METHOD metGetTextListName : STRING
VAR_INPUT
	enTypeOfBacNetFunktionIn		:	enTypeOfBacNetFunktion;
	enTypeOfBacNetTextListIn		:	enTypeOfBacNetTextList;
END_VAR
(* Standart Text *)
IF NOT fbxUseExklTxtList.xValue THEN
	CASE enTypeOfBacNetFunktionIn OF
		(* AT_ANLAGENSCHALTER *)
		enTypeOfBacNetFunktion.Type_Anlagenschalter :
			CASE enTypeOfBacNetTextListIn OF
				enTypeOfBacNetTextList.DESCRIPTION 	:
					metGetTextListName 	:= 'CtaAppBacNetKBOB.TXT_AT_ANLAGENSCHALTER_DESCRIPTION';
				enTypeOfBacNetTextList.ENDING		:
					metGetTextListName 	:= 'CtaAppBacNetKBOB.TXT_AT_ANLAGENSCHALTER_ENDING';
				enTypeOfBacNetTextList.EVENTMESSAGE :
					metGetTextListName 	:= 'CtaAppBacNetKBOB.TXT_AT_ANLAGENSCHALTER_EVENTMESSAGE';
				enTypeOfBacNetTextList.NC			:
					metGetTextListName 	:= 'CtaAppBacNetKBOB.TXT_AT_ANLAGENSCHALTER_NC';
				enTypeOfBacNetTextList.PRESENTVALUE	:
					metGetTextListName	:=	'CtaAppBacNetKBOB.TXT_AT_ANLAGENSCHALTER_PRESV';
				ELSE
					metGetTextListName	:= '';
			END_CASE
		(* AT_ANTRIEB_STETIG *)
		enTypeOfBacNetFunktion.Type_AntriebStetig :
			CASE enTypeOfBacNetTextListIn OF
				enTypeOfBacNetTextList.DESCRIPTION 	:
					metGetTextListName	:= 	'CtaAppBacNetKBOB.TXT_AT_ANTRIEB_STETIG_DESCRIPTION';
				enTypeOfBacNetTextList.ENDING		:
					metGetTextListName	:= 	'CtaAppBacNetKBOB.TXT_AT_ANTRIEB_STETIG_ENDING';
				enTypeOfBacNetTextList.EVENTMESSAGE :
					metGetTextListName	:= 	'CtaAppBacNetKBOB.TXT_AT_ANTRIEB_STETIG_EVENTMESSAGE';
				enTypeOfBacNetTextList.NC			:
					metGetTextListName	:=	'CtaAppBacNetKBOB.TXT_AT_ANTRIEB_STETIG_NC';
				enTypeOfBacNetTextList.PRESENTVALUE	:
					metGetTextListName	:=	'CtaAppBacNetKBOB.TXT_AT_ANTRIEB_STETIG_PRESV';
				ELSE
					metGetTextListName	:= '';
			END_CASE;	
		(* AT_MESSWERTGEBER_BINAR *)
		enTypeOfBacNetFunktion.Type_MesswertgeberBinär :
			CASE enTypeOfBacNetTextListIn OF
				enTypeOfBacNetTextList.DESCRIPTION 	:
					metGetTextListName	:= 	'CtaAppBacNetKBOB.TXT_AT_MESSWERTGEBER_BINAR_DESCRIPTION';
				enTypeOfBacNetTextList.ENDING		:
					metGetTextListName	:= 	'CtaAppBacNetKBOB.TXT_AT_MESSWERTGEBER_BINAR_ENDING';
				enTypeOfBacNetTextList.EVENTMESSAGE :
					metGetTextListName	:= 	'CtaAppBacNetKBOB.TXT_AT_MESSWERTGEBER_BINAR_EVENTMESSAGE';
				enTypeOfBacNetTextList.NC			:
					metGetTextListName	:=	'CtaAppBacNetKBOB.TXT_AT_MESSWERTGEBER_BINAR_NC';
				enTypeOfBacNetTextList.PRESENTVALUE	:
					metGetTextListName	:=	'CtaAppBacNetKBOB.TXT_AT_MESSWERTGEBER_BINAR_PRESV';
				ELSE
					metGetTextListName	:= '';
			END_CASE;
		(* AT_MESSWERTGEBER_STETIG *)
		enTypeOfBacNetFunktion.Type_MesswertgeberStetig :
			CASE enTypeOfBacNetTextListIn OF
				enTypeOfBacNetTextList.DESCRIPTION 	:
					metGetTextListName	:= 	'CtaAppBacNetKBOB.TXT_AT_MESSWERTGEBER_STETIG_DESCRIPTION';
				enTypeOfBacNetTextList.ENDING		:
					metGetTextListName	:= 	'CtaAppBacNetKBOB.TXT_AT_MESSWERTGEBER_STETIG_ENDING';
				enTypeOfBacNetTextList.EVENTMESSAGE :
					metGetTextListName	:= 	'CtaAppBacNetKBOB.TXT_AT_MESSWERTGEBER_STETIG_EVENTMESSAGE';
				enTypeOfBacNetTextList.NC			:
					metGetTextListName	:=	'CtaAppBacNetKBOB.TXT_AT_MESSWERTGEBER_STETIG_NC';
				enTypeOfBacNetTextList.PRESENTVALUE	:
					metGetTextListName	:=	'CtaAppBacNetKBOB.TXT_AT_MESSWERTGEBER_STETIG_PRESV';
				ELSE
					metGetTextListName	:= '';
			END_CASE;
		(* AT_AUTOMATIONSSTATION *)
		enTypeOfBacNetFunktion.Type_Automationsstation :
			CASE enTypeOfBacNetTextListIn OF
				enTypeOfBacNetTextList.DESCRIPTION 	:
					metGetTextListName	:= 	'CtaAppBacNetKBOB.TXT_AT_AUTOMATIONSSTATION_DESCRIPTION';
				enTypeOfBacNetTextList.ENDING		:
					metGetTextListName	:= 	'CtaAppBacNetKBOB.TXT_AT_AUTOMATIONSSTATION_ENDING';
				enTypeOfBacNetTextList.EVENTMESSAGE :
					metGetTextListName	:= 	'CtaAppBacNetKBOB.TXT_AT_AUTOMATIONSSTATION_EVENTMESSAGE';
				enTypeOfBacNetTextList.NC			:
					metGetTextListName	:=	'CtaAppBacNetKBOB.TXT_AT_AUTOMATIONSSTATION_NC';
				enTypeOfBacNetTextList.PRESENTVALUE	:
					metGetTextListName	:=	'CtaAppBacNetKBOB.TXT_AT_AUTOMATIONSSTATION_PRESV';
				ELSE
					metGetTextListName	:= '';
			END_CASE;
		(* AT_ANLAGEFUNKTION *)
		enTypeOfBacNetFunktion.Type_Anlagefunktion :
			CASE enTypeOfBacNetTextListIn OF
				enTypeOfBacNetTextList.DESCRIPTION 	:
					metGetTextListName	:= 	'CtaAppBacNetKBOB.TXT_AT_ANLAGEFUNKTION_DESCRIPTION';
				enTypeOfBacNetTextList.ENDING		:
					metGetTextListName	:= 	'CtaAppBacNetKBOB.TXT_AT_ANLAGEFUNKTION_ENDING';
				enTypeOfBacNetTextList.EVENTMESSAGE :
					metGetTextListName	:= 	'CtaAppBacNetKBOB.TXT_AT_ANLAGEFUNKTION_EVENTMESSAGE';
				enTypeOfBacNetTextList.NC			:
					metGetTextListName	:=	'CtaAppBacNetKBOB.TXT_AT_ANLAGEFUNKTION_NC';
				enTypeOfBacNetTextList.PRESENTVALUE	:
					metGetTextListName	:=	'CtaAppBacNetKBOB.TXT_AT_ANLAGEFUNKTION_PRESV';
				ELSE
					metGetTextListName	:= '';
			END_CASE;		
	ELSE
		metGetTextListName := '';	
	END_CASE;
ELSE
	CASE enTypeOfBacNetFunktionIn OF
		(* AT_ANLAGENSCHALTER *)
		enTypeOfBacNetFunktion.Type_Anlagenschalter :
			CASE enTypeOfBacNetTextListIn OF
				enTypeOfBacNetTextList.DESCRIPTION 	:
					metGetTextListName 	:= 'TXT_AT_ANLAGENSCHALTER_DESCRIPTION';
				enTypeOfBacNetTextList.ENDING		:
					metGetTextListName 	:= 'TXT_AT_ANLAGENSCHALTER_ENDING';
				enTypeOfBacNetTextList.EVENTMESSAGE :
					metGetTextListName 	:= 'TXT_AT_ANLAGENSCHALTER_EVENTMESSAGE';
				enTypeOfBacNetTextList.NC			:
					metGetTextListName 	:= 'TXT_AT_ANLAGENSCHALTER_NC';
				enTypeOfBacNetTextList.PRESENTVALUE	:
					metGetTextListName	:=	'TXT_AT_ANLAGENSCHALTER_PRESV';
				ELSE
					metGetTextListName	:= '';
			END_CASE
		(* AT_ANTRIEB_STETIG *)
		enTypeOfBacNetFunktion.Type_AntriebStetig :
			CASE enTypeOfBacNetTextListIn OF
				enTypeOfBacNetTextList.DESCRIPTION 	:
					metGetTextListName	:= 	'TXT_AT_ANTRIEB_STETIG_DESCRIPTION';
				enTypeOfBacNetTextList.ENDING		:
					metGetTextListName	:= 	'TXT_AT_ANTRIEB_STETIG_ENDING';
				enTypeOfBacNetTextList.EVENTMESSAGE :
					metGetTextListName	:= 	'TXT_AT_ANTRIEB_STETIG_EVENTMESSAGE';
				enTypeOfBacNetTextList.NC			:
					metGetTextListName	:=	'TXT_AT_ANTRIEB_STETIG_NC';
				enTypeOfBacNetTextList.PRESENTVALUE	:
					metGetTextListName	:=	'TXT_AT_ANTRIEB_STETIG_PRESV';
				ELSE
					metGetTextListName	:= '';
			END_CASE;	
		(* AT_MESSWERTGEBER_BINAR *)
		enTypeOfBacNetFunktion.Type_MesswertgeberBinär :
			CASE enTypeOfBacNetTextListIn OF
				enTypeOfBacNetTextList.DESCRIPTION 	:
					metGetTextListName	:= 	'TXT_AT_MESSWERTGEBER_BINAR_DESCRIPTION';
				enTypeOfBacNetTextList.ENDING		:
					metGetTextListName	:= 	'TXT_AT_MESSWERTGEBER_BINAR_ENDING';
				enTypeOfBacNetTextList.EVENTMESSAGE :
					metGetTextListName	:= 	'TXT_AT_MESSWERTGEBER_BINAR_EVENTMESSAGE';
				enTypeOfBacNetTextList.NC			:
					metGetTextListName	:=	'TXT_AT_MESSWERTGEBER_BINAR_NC';
				enTypeOfBacNetTextList.PRESENTVALUE	:
					metGetTextListName	:=	'TXT_AT_MESSWERTGEBER_BINAR_PRESV';
				ELSE
					metGetTextListName	:= '';
			END_CASE;
		(* AT_MESSWERTGEBER_STETIG *)
		enTypeOfBacNetFunktion.Type_MesswertgeberStetig :
			CASE enTypeOfBacNetTextListIn OF
				enTypeOfBacNetTextList.DESCRIPTION 	:
					metGetTextListName	:= 	'TXT_AT_MESSWERTGEBER_STETIG_DESCRIPTION';
				enTypeOfBacNetTextList.ENDING		:
					metGetTextListName	:= 	'TXT_AT_MESSWERTGEBER_STETIG_ENDING';
				enTypeOfBacNetTextList.EVENTMESSAGE :
					metGetTextListName	:= 	'TXT_AT_MESSWERTGEBER_STETIG_EVENTMESSAGE';
				enTypeOfBacNetTextList.NC			:
					metGetTextListName	:=	'TXT_AT_MESSWERTGEBER_STETIG_NC';
				enTypeOfBacNetTextList.PRESENTVALUE	:
					metGetTextListName	:=	'TXT_AT_MESSWERTGEBER_STETIG_PRESV';
				ELSE
					metGetTextListName	:= '';
			END_CASE;
		(* AT_AUTOMATIONSSTATION *)
		enTypeOfBacNetFunktion.Type_Automationsstation :
			CASE enTypeOfBacNetTextListIn OF
				enTypeOfBacNetTextList.DESCRIPTION 	:
					metGetTextListName	:= 	'TXT_AT_AUTOMATIONSSTATION_DESCRIPTION';
				enTypeOfBacNetTextList.ENDING		:
					metGetTextListName	:= 	'TXT_AT_AUTOMATIONSSTATION_ENDING';
				enTypeOfBacNetTextList.EVENTMESSAGE :
					metGetTextListName	:= 	'TXT_AT_MESSWERTGEBER_STETIG_EVENTMESSAGE';
				enTypeOfBacNetTextList.NC			:
					metGetTextListName	:=	'TXT_AT_MESSWERTGEBER_STETIG_NC';
				enTypeOfBacNetTextList.PRESENTVALUE	:
					metGetTextListName	:=	'TXT_AT_MESSWERTGEBER_STETIG_PRESV';
				ELSE
					metGetTextListName	:= '';
			END_CASE;
		(* AT_ANLAGEFUNKTION *)
		enTypeOfBacNetFunktion.Type_Anlagefunktion :
			CASE enTypeOfBacNetTextListIn OF
				enTypeOfBacNetTextList.DESCRIPTION 	:
					metGetTextListName	:= 	'TXT_AT_ANLAGEFUNKTION_DESCRIPTION';
				enTypeOfBacNetTextList.ENDING		:
					metGetTextListName	:= 	'TXT_AT_ANLAGEFUNKTION_ENDING';
				enTypeOfBacNetTextList.EVENTMESSAGE :
					metGetTextListName	:= 	'TXT_AT_ANLAGEFUNKTION_EVENTMESSAGE';
				enTypeOfBacNetTextList.NC			:
					metGetTextListName	:=	'TXT_AT_ANLAGEFUNKTION_NC';
				enTypeOfBacNetTextList.PRESENTVALUE	:
					metGetTextListName	:=	'TXT_AT_ANLAGEFUNKTION_PRESV';
				ELSE
					metGetTextListName	:= '';
			END_CASE;		
	ELSE
		metGetTextListName := '';	
	END_CASE;
END_IF;
END_METHOD

PROPERTY proKBOB_REV : enKBOB_REV
GET
proKBOB_REV := fbenBacNetKbobRev.proValue;
END_GET
END_PROPERTY

PROPERTY P_fbenBacNetKbobRev : CtaSysConfig.ITF_INT
GET
P_fbenBacNetKbobRev := fbenBacNetKbobRev;
END_GET
END_PROPERTY

PROPERTY P_fbxEnableBacNet : CtaSysConfig.ITF_BOOL
GET
P_fbxEnableBacNet := fbxEnableBacNet;
END_GET
END_PROPERTY

PROPERTY P_fbxUseAKS : CtaSysConfig.ITF_BOOL
GET
P_fbxUseAKS := fbxUseAKS;
END_GET
END_PROPERTY

PROPERTY P_fbxUseExklTxtList : CtaSysConfig.ITF_BOOL
GET
P_fbxUseExklTxtList := fbxUseExklTxtList;
END_GET
END_PROPERTY

PROPERTY proTimeToOnline : TIME
GET
IF TON_DELAY_START.Q AND uiCountCreatetObj >= uiCountObj THEN
	proTimeToOnline := T#0S;
ELSE
	proTimeToOnline := (TON_DELAY_START.PT - TON_DELAY_START.ET) + ((uiCountObj * T#6S) - (uiCountCreatetObj * T#6S));
END_IF
END_GET
END_PROPERTY

PROPERTY proDestroyBacNetOverrideXmlNode : BOOL
GET
proDestroyBacNetOverrideXmlNode := xDestroyBacNetOverrideNode;
END_GET
END_PROPERTY

PROPERTY proRebootRequired : BOOL
SET
xRebootRequired := proRebootRequired;
END_SET
GET
proRebootRequired := xRebootRequired;
END_GET
END_PROPERTY

METHOD metAddObj
VAR_INPUT
	ITF_OBJ				:	ITF_OBJ_ID_BASE;
END_VAR
IF __QUERYINTERFACE(ITF_OBJ,ITF_OBJ) THEN
	IF __QUERYINTERFACE(ITF_FIRST_OBJ,ITF_FIRST_OBJ) THEN
		IF ITF_FIRST_OBJ.proINextObj = 0 THEN
			ITF_FIRST_OBJ.proINextObj := ITF_OBJ;
		END_IF;
		IF __QUERYINTERFACE(ITF_NEXT_OBJ,ITF_NEXT_OBJ) THEN
			ITF_NEXT_OBJ.proINextObj := ITF_OBJ;
			ITF_NEXT_OBJ := ITF_OBJ;
		ELSE
			ITF_NEXT_OBJ := ITF_OBJ;
		END_IF;
	ELSIF ITF_FIRST_OBJ = 0 THEN
		ITF_FIRST_OBJ := ITF_OBJ;
	END_IF;	
	uiCountObj := uiCountObj + 1;
END_IF
END_METHOD

ACTION BACNETLIBPARACHECK:
{IF defined (variable: WagoTypesBACnet.Parameter.LEN_BACnetDescription)}
	{IF defined (task: PLC_PRG_Task)}
		{ IF hasconstantvalue(WagoTypesBACnet.Parameter.LEN_BACnetDescription,128,<>)}
			{error 'WagoTypesBACnet.Parameter.LEN_BACnetDescription value <> 128'}
		{END_IF}
	{ELSE}
		{info 'CtaAppBacNetKBOB wurde als Bibliothek Compiliert'}
	{END_IF}
{ELSE}
	{error 'WagoTypesBACnet.Parameter.LEN_BACnetDescription not existing'}
{END_IF}
END_ACTION

PROPERTY P_fbdiDeviceId : CtaSysConfig.ITF_DINT
GET
P_fbdiDeviceId := fbdiDeviceId;
END_GET
END_PROPERTY

PROPERTY P_fbxAnsiCodiert : CtaSysConfig.ITF_BOOL
GET
P_fbxAnsiCodiert := fbxAnsiCodiert;
END_GET
END_PROPERTY

END_FUNCTION_BLOCK

// 30 Program Organization Units/FCs/BacNetIni/fcBacNetIni
FUNCTION fcBacNetIni : BOOL
VAR_INPUT
END_VAR
VAR
	stCommand			:	STRING(255);
	RTS_IEC_RESULT		:	SysTypes.RTS_IEC_RESULT;
END_VAR

(* Replace the persistence-delete from false to true *)
stCommand := 'sed -i $'s/persistence-delete=false/persistence-delete=true/$' /home/user/bacnet/config/bacconfig.ini';
SysProcess_Implementation.SysProcessExecuteCommand(stCommand,ADR(RTS_IEC_RESULT));

END_FUNCTION

// 21 Interface/BACNET_PARAMETER/ITF_BACNET_PARAMETER
INTERFACE ITF_BACNET_PARAMETER EXTENDS __System.IQueryinterface

METHOD metGetTextListName : STRING
VAR_INPUT
	enTypeOfBacNetFunktionIn		:	enTypeOfBacNetFunktion;
	enTypeOfBacNetTextListIn		:	enTypeOfBacNetTextList;
END_VAR
END_METHOD

METHOD metRequestDelete : BOOL
END_METHOD

PROPERTY proCreate : Bool
GET
END_GET
END_PROPERTY

PROPERTY proDelete : Bool
GET
END_GET
END_PROPERTY

PROPERTY proInitDone : BOOL
GET
END_GET
END_PROPERTY

PROPERTY proKBOB_REV : enKBOB_REV
GET
END_GET
END_PROPERTY

PROPERTY proUseAKS : BOOL
GET
END_GET
END_PROPERTY

PROPERTY P_fbxEnableBacNet : CtaSysConfig.ITF_BOOL
GET
END_GET
END_PROPERTY

PROPERTY P_fbxUseAKS : CtaSysConfig.ITF_BOOL
GET
END_GET
END_PROPERTY

PROPERTY P_fbxUseExklTxtList : CtaSysConfig.ITF_BOOL
GET
END_GET
END_PROPERTY

PROPERTY P_fbenBacNetKbobRev : CtaSysConfig.ITF_INT
GET
END_GET
END_PROPERTY

PROPERTY proTimeToOnline : TIME
GET
END_GET
END_PROPERTY

METHOD metAddObj
VAR_INPUT
	ITF_OBJ				:	ITF_OBJ_ID_BASE;
END_VAR
END_METHOD

PROPERTY proRebootRequired : BOOL
SET
END_SET
GET
END_GET
END_PROPERTY

PROPERTY proDestroyBacNetOverrideXmlNode : BOOL
GET
END_GET
END_PROPERTY

PROPERTY P_fbdiDeviceId : CtaSysConfig.ITF_DINT
GET
END_GET
END_PROPERTY

PROPERTY P_fbxAnsiCodiert : CtaSysConfig.ITF_BOOL
GET
END_GET
END_PROPERTY

END_INTERFACE

// 30 Program Organization Units/Pou/BAC_NET
PROGRAM BAC_NET
VAR
END_VAR

(* PARAMETER *)
GVL_BACNET.fbBacNetParameter();
(* AT_DEVICE *)
GVL_BACNET.fbAtAutomationsstation();

END_PROGRAM

// 30 Program Organization Units/FBs/AT_FUNKTIONEN/AT_AUTOMATIONSTATION/FB_AT_AUTOMATIONSSTATION
FUNCTION_BLOCK FB_AT_AUTOMATIONSSTATION EXTENDS FB_OBJ_ID_BASE
VAR
	(* BacNet Objects *)
	A_DV_1				:	WagoSysBACnet.FbDevice_small(-1);						// Device
	B_CL_1				:	WagoSysBACnet.FbCalendar_large(-1);                     // Kalender variable Feiertage
	C_CL_2				:	WagoSysBACnet.FbCalendar_large(-1);                     // Kalender Halbe Tage
	D_CL_3				:	WagoSysBACnet.FbCalendar_large(-1);                     // Kalender feste Feiertage
	E_CL_4				:	WagoSysBACnet.FbCalendar_large(-1);                     // Kalender Ferien
	F_EL_1				:	WagoSysBACnet.FbEventLog_large(-1);						// Eventlog
	G_NC_1				:	WagoSysBACnet.FbNotificationClass_large(-1);			// Notification Class  1 Group Sicherheitsalarm
	G_NC_2				:	WagoSysBACnet.FbNotificationClass_large(-1);			// Notification Class  2 Group Sicherheitsalarm
	G_NC_3				:	WagoSysBACnet.FbNotificationClass_large(-1);			// Notification Class  3 Group Sicherheitsalarm
	G_NC_4				:	WagoSysBACnet.FbNotificationClass_large(-1);			// Notification Class  4 Group Sicherheitsalarm
	H_NC_32				:	WagoSysBACnet.FbNotificationClass_large(-1);			// Notification Class 32 Group Sicherheitsalarm
	H_NC_33				:	WagoSysBACnet.FbNotificationClass_large(-1);			// Notification Class 33 Group Sicherheitsalarm
	H_NC_34				:	WagoSysBACnet.FbNotificationClass_large(-1);			// Notification Class 34 Group Sicherheitsalarm
	H_NC_35				:	WagoSysBACnet.FbNotificationClass_large(-1);			// Notification Class 35 Group Sicherheitsalarm
	I_NC_64				:	WagoSysBACnet.FbNotificationClass_large(-1);			// Notification Class 64 Group Sicherheitsalarm
	I_NC_65				:	WagoSysBACnet.FbNotificationClass_large(-1);			// Notification Class 65 Group Sicherheitsalarm
	I_NC_66				:	WagoSysBACnet.FbNotificationClass_large(-1);			// Notification Class 66 Group Sicherheitsalarm
	I_NC_67				:	WagoSysBACnet.FbNotificationClass_large(-1);			// Notification Class 67 Group Sicherheitsalarm
	J_NC_96				:	WagoSysBACnet.FbNotificationClass_large(-1);			// Notification Class 96 Group Sicherheitsalarm
	J_NC_97				:	WagoSysBACnet.FbNotificationClass_large(-1);			// Notification Class 97 Group Sicherheitsalarm
	J_NC_98				:	WagoSysBACnet.FbNotificationClass_large(-1);			// Notification Class 98 Group Sicherheitsalarm
	J_NC_99				:	WagoSysBACnet.FbNotificationClass_large(-1);			// Notification Class 99 Group Sicherheitsalarm
	K_NC_128			:	WagoSysBACnet.FbNotificationClass_large(-1);			// Notification Class 128 Group Sicherheitsalarm
	K_NC_129			:	WagoSysBACnet.FbNotificationClass_large(-1);			// Notification Class 129 Group Sicherheitsalarm
	K_NC_130			:	WagoSysBACnet.FbNotificationClass_large(-1);			// Notification Class 130 Group Sicherheitsalarm
	K_NC_131			:	WagoSysBACnet.FbNotificationClass_large(-1);			// Notification Class 131 Group Sicherheitsalarm
	L_NC_160			:	WagoSysBACnet.FbNotificationClass_large(-1);			// Notification Class 160 Group Sicherheitsalarm
	L_NC_161			:	WagoSysBACnet.FbNotificationClass_large(-1);			// Notification Class 161 Group Sicherheitsalarm
	L_NC_162			:	WagoSysBACnet.FbNotificationClass_large(-1);			// Notification Class 162 Group Sicherheitsalarm
	L_NC_163			:	WagoSysBACnet.FbNotificationClass_large(-1);			// Notification Class 163 Group Sicherheitsalarm
	M_NC_192			:	WagoSysBACnet.FbNotificationClass_large(-1);			// Notification Class 192 Group Sicherheitsalarm
	M_NC_193			:	WagoSysBACnet.FbNotificationClass_large(-1);			// Notification Class 193 Group Sicherheitsalarm
	N_NC_224			:	WagoSysBACnet.FbNotificationClass_large(-1);			// Notification Class 224 Group Sicherheitsalarm
	N_NC_225			:	WagoSysBACnet.FbNotificationClass_large(-1);			// Notification Class 225 Group Sicherheitsalarm	
	O_BV_1				:	WagoSysBACnet.FbBinaryValue_large(-1);					// CPU State
	P_BV_2				:	WagoSysBACnet.FbBinaryValue_large(-1);					// I/O State
	Q_BV_3				:	WagoSysBACnet.FbBinaryValue_large(-1);					// I/O Hand
	R_BV_4				:	WagoSysBACnet.FbBinaryValue_large(-1);					// Heartbeat
	S_BV_5				:	WagoSysBACnet.FbBinaryValue_large(-1);					// BacStack State
	
END_VAR
VAR CONSTANT
	usiAnzBacNetObj	:	USINT	:= 39;
END_VAR

(* Call Base FB*)
SUPER^();
(* Cyclic Action *)
IF xCreatet THEN
	(* DESCTIPTION FIX *)
	metCYCLIC_DESCRIPTION_FIX();
	(* Get Revision *)
	CASE GVL_BACNET.fbBacNetParameter.proKBOB_REV OF
		(* KBOB 2021 V2 *)
		enKBOB_REV.KBOB_REV2021_V2:
			metCYCLIC_KBOB_2021_V2();
		(* KBOB 2017 V1 *)
		enKBOB_REV.KBOB_REV2017_V1:
			metCYCLIC_KBOB_2017_V1();
		(* Default *)
		ELSE
			metCYCLIC_KBOB_2021_V2();
	END_CASE;	
END_IF;

METHOD metCYCLIC_KBOB_2017_V1
VAR_INPUT
END_VAR
(* CPU Overload *)
IF O_BV_1.xIsCreated THEN
	O_BV_1.xPresentValue := WagoSysBACnet.Common.ControllerInfo.ILedStatus.eLedStatus = WagoTypesBACnet.eBACnetLedStatus.LED_BT_WARNING_OVERLOAD;
END_IF;

(* Check if CtaSysIO exist *)
{IF defined (variable:CtaSysIO.GVL_IO.fbIO_Manager.xError) AND defined (variable:CtaSysIO.GVL_IO.fbIO_Manager.xHand)}
	(* I/O State*) 
	IF P_BV_2.xIsCreated THEN
		P_BV_2.xPresentValue := CtaSysIO.GVL_IO.fbIO_Manager.xError;
	END_IF;

(* I/O Hand *)
	IF Q_BV_3.xIsCreated THEN
		Q_BV_3.xPresentValue := CtaSysIO.GVL_IO.fbIO_Manager.xHand;
	END_IF
{ELSE}
	{warning 'FB_AUTOMATIONSSTATION I/O Infos only with CtaSysIO Library'}
{END_IF}

(* BacStack Error *)
IF S_BV_5.xIsCreated THEN
	S_BV_5.xPresentValue := WagoSysBACnet.Common.ControllerInfo.ILedStatus.eLedStatus = WagoTypesBACnet.eBACnetLedStatus.LED_BT_ERROR_INTERNAL;
END_IF;
END_METHOD

METHOD metCYCLIC_KBOB_2021_V2
VAR_INPUT
END_VAR
(* CPU Overload *)
IF O_BV_1.xIsCreated THEN
	O_BV_1.xPresentValue := WagoSysBACnet.Common.ControllerInfo.ILedStatus.eLedStatus = WagoTypesBACnet.eBACnetLedStatus.LED_BT_WARNING_OVERLOAD;
END_IF;

(* Check if CtaSysIO exist *)
{IF defined (variable:CtaSysIO.GVL_IO.fbIO_Manager.xError) AND defined (variable:CtaSysIO.GVL_IO.fbIO_Manager.xHand)}
	(* I/O State*) 
	IF P_BV_2.xIsCreated THEN
		P_BV_2.xPresentValue := CtaSysIO.GVL_IO.fbIO_Manager.xError;
	END_IF;

(* I/O Hand *)
	IF Q_BV_3.xIsCreated THEN
		Q_BV_3.xPresentValue := CtaSysIO.GVL_IO.fbIO_Manager.xHand;
	END_IF
{ELSE}
	{warning 'FB_AUTOMATIONSSTATION I/O Infos only with CtaSysIO Library'}
{END_IF}

(* BacStack Error *)
IF S_BV_5.xIsCreated THEN
	S_BV_5.xPresentValue := WagoSysBACnet.Common.ControllerInfo.ILedStatus.eLedStatus = WagoTypesBACnet.eBACnetLedStatus.LED_BT_ERROR_INTERNAL;
END_IF;
END_METHOD

METHOD metCYCLIC_DESCRIPTION_FIX
VAR_INPUT
END_VAR
(* A_DV_1 *)
IF A_DV_1.xIsCreated THEN
	IF A_DV_1.sDescription <> A_DV_1._sDescription THEN
		A_DV_1.sDescription := A_DV_1._sDescription;
	END_IF;
END_IF;

(* B_CL_1 *)
IF B_CL_1.xIsCreated THEN
	IF B_CL_1.sDescription <> B_CL_1._sDescription THEN
		B_CL_1.sDescription := B_CL_1._sDescription;
	END_IF;
END_IF;

(* C_CL_2 *)
IF C_CL_2.xIsCreated THEN
	IF C_CL_2.sDescription <> C_CL_2._sDescription THEN
		C_CL_2.sDescription := C_CL_2._sDescription;
	END_IF;
END_IF;

(* D_CL_3 *)
IF D_CL_3.xIsCreated THEN
	IF D_CL_3.sDescription <> D_CL_3._sDescription THEN
		D_CL_3.sDescription := D_CL_3._sDescription;
	END_IF;
END_IF;

(* E_CL_4 *)
IF E_CL_4.xIsCreated THEN
	IF E_CL_4.sDescription <> E_CL_4._sDescription THEN
		E_CL_4.sDescription := E_CL_4._sDescription;
	END_IF;
END_IF;

(* F_EL_1 *)
IF F_EL_1.xIsCreated THEN
	IF F_EL_1.sDescription <> F_EL_1._sDescription THEN
		F_EL_1.sDescription := F_EL_1._sDescription;
	END_IF;
END_IF;

(* G_NC_1 *)
IF G_NC_1.xIsCreated THEN
	IF G_NC_1.sDescription <> G_NC_1._sDescription THEN
		G_NC_1.sDescription := G_NC_1._sDescription;
	END_IF;
END_IF;

(* G_NC_2 *)
IF G_NC_2.xIsCreated THEN
	IF G_NC_2.sDescription <> G_NC_2._sDescription THEN
		G_NC_2.sDescription := G_NC_2._sDescription;
	END_IF;
END_IF;

(* G_NC_3 *)
IF G_NC_3.xIsCreated THEN
	IF G_NC_3.sDescription <> G_NC_3._sDescription THEN
		G_NC_3.sDescription := G_NC_3._sDescription;
	END_IF;
END_IF;

(* G_NC_4 *)
IF G_NC_4.xIsCreated THEN
	IF G_NC_4.sDescription <> G_NC_4._sDescription THEN
		G_NC_4.sDescription := G_NC_4._sDescription;
	END_IF;
END_IF;

(* H_NC_32 *)
IF H_NC_32.xIsCreated THEN
	IF H_NC_32.sDescription <> H_NC_32._sDescription THEN
		H_NC_32.sDescription := H_NC_32._sDescription;
	END_IF;
END_IF;

(* H_NC_33 *)
IF H_NC_33.xIsCreated THEN
	IF H_NC_33.sDescription <> H_NC_33._sDescription THEN
		H_NC_33.sDescription := H_NC_33._sDescription;
	END_IF;
END_IF;

(* H_NC_34 *)
IF H_NC_34.xIsCreated THEN
	IF H_NC_34.sDescription <> H_NC_34._sDescription THEN
		H_NC_34.sDescription := H_NC_34._sDescription;
	END_IF;
END_IF;

(* H_NC_35 *)
IF H_NC_35.xIsCreated THEN
	IF H_NC_35.sDescription <> H_NC_35._sDescription THEN
		H_NC_35.sDescription := H_NC_35._sDescription;
	END_IF;
END_IF;

(* I_NC_64 *)
IF I_NC_64.xIsCreated THEN
	IF I_NC_64.sDescription <> I_NC_64._sDescription THEN
		I_NC_64.sDescription := I_NC_64._sDescription;
	END_IF;
END_IF;

(* I_NC_65 *)
IF I_NC_65.xIsCreated THEN
	IF I_NC_65.sDescription <> I_NC_65._sDescription THEN
		I_NC_65.sDescription := I_NC_65._sDescription;
	END_IF;
END_IF;

(* I_NC_66 *)
IF I_NC_66.xIsCreated THEN
	IF I_NC_66.sDescription <> I_NC_66._sDescription THEN
		I_NC_66.sDescription := I_NC_66._sDescription;
	END_IF;
END_IF;

(* I_NC_67 *)
IF I_NC_67.xIsCreated THEN
	IF I_NC_67.sDescription <> I_NC_67._sDescription THEN
		I_NC_67.sDescription := I_NC_67._sDescription;
	END_IF;
END_IF;

(* J_NC_96 *)
IF J_NC_96.xIsCreated THEN
	IF J_NC_96.sDescription <> J_NC_96._sDescription THEN
		J_NC_96.sDescription := J_NC_96._sDescription;
	END_IF;
END_IF;

(* J_NC_97 *)
IF J_NC_97.xIsCreated THEN
	IF J_NC_97.sDescription <> J_NC_97._sDescription THEN
		J_NC_97.sDescription := J_NC_97._sDescription;
	END_IF;
END_IF;

(* J_NC_98 *)
IF J_NC_98.xIsCreated THEN
	IF J_NC_98.sDescription <> J_NC_98._sDescription THEN
		J_NC_98.sDescription := J_NC_98._sDescription;
	END_IF;
END_IF;

(* J_NC_99 *)
IF J_NC_99.xIsCreated THEN
	IF J_NC_99.sDescription <> J_NC_99._sDescription THEN
		J_NC_99.sDescription := J_NC_99._sDescription;
	END_IF;
END_IF;

(* K_NC_128 *)
IF K_NC_128.xIsCreated THEN
	IF K_NC_128.sDescription <> K_NC_128._sDescription THEN
		K_NC_128.sDescription := K_NC_128._sDescription;
	END_IF;
END_IF;

(* K_NC_129 *)
IF K_NC_129.xIsCreated THEN
	IF K_NC_129.sDescription <> K_NC_129._sDescription THEN
		K_NC_129.sDescription := K_NC_129._sDescription;
	END_IF;
END_IF;

(* K_NC_130 *)
IF K_NC_130.xIsCreated THEN
	IF K_NC_130.sDescription <> K_NC_130._sDescription THEN
		K_NC_130.sDescription := K_NC_130._sDescription;
	END_IF;
END_IF;

(* K_NC_131 *)
IF K_NC_131.xIsCreated THEN
	IF K_NC_131.sDescription <> K_NC_131._sDescription THEN
		K_NC_131.sDescription := K_NC_131._sDescription;
	END_IF;
END_IF;

(* L_NC_160 *)
IF L_NC_160.xIsCreated THEN
	IF L_NC_160.sDescription <> L_NC_160._sDescription THEN
		L_NC_160.sDescription := L_NC_160._sDescription;
	END_IF;
END_IF;

(* L_NC_161 *)
IF L_NC_161.xIsCreated THEN
	IF L_NC_161.sDescription <> L_NC_161._sDescription THEN
		L_NC_161.sDescription := L_NC_161._sDescription;
	END_IF;
END_IF;

(* L_NC_162 *)
IF L_NC_162.xIsCreated THEN
	IF L_NC_162.sDescription <> L_NC_162._sDescription THEN
		L_NC_162.sDescription := L_NC_162._sDescription;
	END_IF;
END_IF;

(* L_NC_163 *)
IF L_NC_163.xIsCreated THEN
	IF L_NC_163.sDescription <> L_NC_163._sDescription THEN
		L_NC_163.sDescription := L_NC_163._sDescription;
	END_IF;
END_IF;

(* M_NC_192 *)
IF M_NC_192.xIsCreated THEN
	IF M_NC_192.sDescription <> M_NC_192._sDescription THEN
		M_NC_192.sDescription := M_NC_192._sDescription;
	END_IF;
END_IF;

(* M_NC_193 *)
IF M_NC_193.xIsCreated THEN
	IF M_NC_193.sDescription <> M_NC_193._sDescription THEN
		M_NC_193.sDescription := M_NC_193._sDescription;
	END_IF;
END_IF;

(* N_NC_224 *)
IF N_NC_224.xIsCreated THEN
	IF N_NC_224.sDescription <> N_NC_224._sDescription THEN
		N_NC_224.sDescription := N_NC_224._sDescription;
	END_IF;
END_IF;

(* N_NC_225 *)
IF N_NC_225.xIsCreated THEN
	IF N_NC_225.sDescription <> N_NC_225._sDescription THEN
		N_NC_225.sDescription := N_NC_225._sDescription;
	END_IF;
END_IF;

(* O_BV_1 *)
IF O_BV_1.xIsCreated THEN
	IF O_BV_1.sDescription <> O_BV_1._sDescription THEN
		O_BV_1.sDescription := O_BV_1._sDescription;
	END_IF;
END_IF;

(* P_BV_2 *)
IF P_BV_2.xIsCreated THEN
	IF P_BV_2.sDescription <> P_BV_2._sDescription THEN
		P_BV_2.sDescription := P_BV_2._sDescription;
	END_IF;
END_IF;

(* Q_BV_3 *)
IF Q_BV_3.xIsCreated THEN
	IF Q_BV_3.sDescription <> Q_BV_3._sDescription THEN
		Q_BV_3.sDescription := Q_BV_3._sDescription;
	END_IF;
END_IF;

(* R_BV_4 *)
IF R_BV_4.xIsCreated THEN
	IF R_BV_4.sDescription <> R_BV_4._sDescription THEN
		R_BV_4.sDescription := R_BV_4._sDescription;
	END_IF;
END_IF;

(* S_BV_5 *)
IF S_BV_5.xIsCreated THEN
	IF S_BV_5.sDescription <> S_BV_5._sDescription THEN
		S_BV_5.sDescription := S_BV_5._sDescription;
	END_IF;
END_IF;
END_METHOD

(*FB_Exit muss explizit implementiert werden. Wenn es eine Implementierung gibt, dann wird 
die Methode aufgerufen, bevor die Steuerung den Code der Funktionsbaustein-Instanz entfernt
(impliziter Aufruf. Der Rückgabewert wird nicht ausgewertet.*)
METHOD FB_Exit : BOOL
VAR_INPUT
	(* TRUE: Die Exit-Methode wird aufgerufen, um die Instanz zu verlassen, die hinterher kopiert wird Online-Change).  *)
	bInCopyCode	: BOOL;
END_VAR
(* A_DV_1 *)
IF A_DV_1.xIsCreated THEN
	A_DV_1.Delete();
END_IF;

(* B_CL_1 *)
IF B_CL_1.xIsCreated THEN
	B_CL_1.Delete();
END_IF;

(* C_CL_2 *)
IF C_CL_2.xIsCreated THEN
	C_CL_2.Delete();
END_IF;

(* D_CL_3 *)
IF D_CL_3.xIsCreated THEN
	D_CL_3.Delete();
END_IF;

(* E_CL_4 *)
IF E_CL_4.xIsCreated THEN
	E_CL_4.Delete();
END_IF;

(* F_EL_1 *)
IF F_EL_1.xIsCreated THEN
	F_EL_1.Delete();
END_IF;

(* G_NC_1 *)
IF G_NC_1.xIsCreated THEN
	G_NC_1.Delete();
END_IF;

(* G_NC_2 *)
IF G_NC_2.xIsCreated THEN
	G_NC_2.Delete();
END_IF;

(* G_NC_3 *)
IF G_NC_3.xIsCreated THEN
	G_NC_3.Delete();
END_IF;

(* G_NC_4 *)
IF G_NC_4.xIsCreated THEN
	G_NC_4.Delete();
END_IF;

(* H_NC_32 *)
IF H_NC_32.xIsCreated THEN
	H_NC_32.Delete();
END_IF;

(* H_NC_33 *)
IF H_NC_33.xIsCreated THEN
	H_NC_33.Delete();
END_IF;

(* H_NC_34 *)
IF H_NC_34.xIsCreated THEN
	H_NC_34.Delete();
END_IF;

(* H_NC_35 *)
IF H_NC_35.xIsCreated THEN
	H_NC_35.Delete();
END_IF;

(* I_NC_64 *)
IF I_NC_64.xIsCreated THEN
	I_NC_64.Delete();
END_IF;

(* I_NC_65 *)
IF I_NC_65.xIsCreated THEN
	I_NC_65.Delete();
END_IF;

(* I_NC_66 *)
IF I_NC_66.xIsCreated THEN
	I_NC_66.Delete();
END_IF;

(* I_NC_67 *)
IF I_NC_67.xIsCreated THEN
	I_NC_67.Delete();
END_IF;

(* J_NC_96 *)
IF J_NC_96.xIsCreated THEN
	J_NC_96.Delete();
END_IF;

(* J_NC_97 *)
IF J_NC_97.xIsCreated THEN
	J_NC_97.Delete();
END_IF;

(* J_NC_98 *)
IF J_NC_98.xIsCreated THEN
	J_NC_98.Delete();
END_IF;

(* J_NC_99 *)
IF J_NC_99.xIsCreated THEN
	J_NC_99.Delete();
END_IF;

(* K_NC_128 *)
IF K_NC_128.xIsCreated THEN
	K_NC_128.Delete();
END_IF;

(* K_NC_129 *)
IF K_NC_129.xIsCreated THEN
	K_NC_129.Delete();
END_IF;

(* K_NC_130 *)
IF K_NC_130.xIsCreated THEN
	K_NC_130.Delete();
END_IF;

(* K_NC_131 *)
IF K_NC_131.xIsCreated THEN
	K_NC_131.Delete();
END_IF;

(* L_NC_160 *)
IF L_NC_160.xIsCreated THEN
	L_NC_160.Delete();
END_IF;

(* L_NC_161 *)
IF L_NC_161.xIsCreated THEN
	L_NC_161.Delete();
END_IF;

(* L_NC_162 *)
IF L_NC_162.xIsCreated THEN
	L_NC_162.Delete();
END_IF;

(* L_NC_163 *)
IF L_NC_163.xIsCreated THEN
	L_NC_163.Delete();
END_IF;

(* M_NC_192 *)
IF M_NC_192.xIsCreated THEN
	M_NC_192.Delete();
END_IF;

(* M_NC_193 *)
IF M_NC_193.xIsCreated THEN
	M_NC_193.Delete();
END_IF;

(* N_NC_224 *)
IF N_NC_224.xIsCreated THEN
	N_NC_224.Delete();
END_IF;

(* N_NC_225 *)
IF N_NC_225.xIsCreated THEN
	N_NC_225.Delete();
END_IF;

(* O_BV_1 *)
IF O_BV_1.xIsCreated THEN
	O_BV_1.Delete();
END_IF;

(* P_BV_2 *)
IF P_BV_2.xIsCreated THEN
	P_BV_2.Delete();
END_IF;

(* Q_BV_3 *)
IF Q_BV_3.xIsCreated THEN
	Q_BV_3.Delete();
END_IF;

(* R_BV_4 *)
IF R_BV_4.xIsCreated THEN
	R_BV_4.Delete();
END_IF;

(* S_BV_5 *)
IF S_BV_5.xIsCreated THEN
	S_BV_5.Delete();
END_IF;
END_METHOD

METHOD metDELETE : BOOL
VAR_INPUT
END_VAR
VAR
	oStatus		:	WagoSysErrorBase.FbResult;
END_VAR
(* A_DV_1 *)
IF A_DV_1.xIsCreated THEN
	A_DV_1.Delete();
END_IF;

(* B_CL_1 *)
IF B_CL_1.xIsCreated THEN
	B_CL_1.Delete();
END_IF;

(* C_CL_2 *)
IF C_CL_2.xIsCreated THEN
	C_CL_2.Delete();
END_IF;

(* D_CL_3 *)
IF D_CL_3.xIsCreated THEN
	D_CL_3.Delete();
END_IF;

(* E_CL_4 *)
IF E_CL_4.xIsCreated THEN
	E_CL_4.Delete();
END_IF;

(* F_EL_1 *)
IF F_EL_1.xIsCreated THEN
	F_EL_1.Delete();
END_IF;

(* G_NC_1 *)
IF G_NC_1.xIsCreated THEN
	G_NC_1.Delete();
END_IF;

(* G_NC_2 *)
IF G_NC_2.xIsCreated THEN
	G_NC_2.Delete();
END_IF;

(* G_NC_3 *)
IF G_NC_3.xIsCreated THEN
	G_NC_3.Delete();
END_IF;

(* G_NC_4 *)
IF G_NC_4.xIsCreated THEN
	G_NC_4.Delete();
END_IF;

(* H_NC_32 *)
IF H_NC_32.xIsCreated THEN
	H_NC_32.Delete();
END_IF;

(* H_NC_33 *)
IF H_NC_33.xIsCreated THEN
	H_NC_33.Delete();
END_IF;

(* H_NC_34 *)
IF H_NC_34.xIsCreated THEN
	H_NC_34.Delete();
END_IF;

(* H_NC_35 *)
IF H_NC_35.xIsCreated THEN
	H_NC_35.Delete();
END_IF;

(* I_NC_64 *)
IF I_NC_64.xIsCreated THEN
	I_NC_64.Delete();
END_IF;

(* I_NC_65 *)
IF I_NC_65.xIsCreated THEN
	I_NC_65.Delete();
END_IF;

(* I_NC_66 *)
IF I_NC_66.xIsCreated THEN
	I_NC_66.Delete();
END_IF;

(* I_NC_67 *)
IF I_NC_67.xIsCreated THEN
	I_NC_67.Delete();
END_IF;

(* J_NC_96 *)
IF J_NC_96.xIsCreated THEN
	J_NC_96.Delete();
END_IF;

(* J_NC_97 *)
IF J_NC_97.xIsCreated THEN
	J_NC_97.Delete();
END_IF;

(* J_NC_98 *)
IF J_NC_98.xIsCreated THEN
	J_NC_98.Delete();
END_IF;

(* J_NC_99 *)
IF J_NC_99.xIsCreated THEN
	J_NC_99.Delete();
END_IF;

(* K_NC_128 *)
IF K_NC_128.xIsCreated THEN
	K_NC_128.Delete();
END_IF;

(* K_NC_129 *)
IF K_NC_129.xIsCreated THEN
	K_NC_129.Delete();
END_IF;

(* K_NC_130 *)
IF K_NC_130.xIsCreated THEN
	K_NC_130.Delete();
END_IF;

(* K_NC_131 *)
IF K_NC_131.xIsCreated THEN
	K_NC_131.Delete();
END_IF;

(* L_NC_160 *)
IF L_NC_160.xIsCreated THEN
	L_NC_160.Delete();
END_IF;

(* L_NC_161 *)
IF L_NC_161.xIsCreated THEN
	L_NC_161.Delete();
END_IF;

(* L_NC_162 *)
IF L_NC_162.xIsCreated THEN
	L_NC_162.Delete();
END_IF;

(* L_NC_163 *)
IF L_NC_163.xIsCreated THEN
	L_NC_163.Delete();
END_IF;

(* M_NC_192 *)
IF M_NC_192.xIsCreated THEN
	M_NC_192.Delete();
END_IF;

(* M_NC_193 *)
IF M_NC_193.xIsCreated THEN
	M_NC_193.Delete();
END_IF;

(* N_NC_224 *)
IF N_NC_224.xIsCreated THEN
	N_NC_224.Delete();
END_IF;

(* N_NC_225 *)
IF N_NC_225.xIsCreated THEN
	N_NC_225.Delete();
END_IF;

(* O_BV_1 *)
IF O_BV_1.xIsCreated THEN
	O_BV_1.Delete();
END_IF;

(* P_BV_2 *)
IF P_BV_2.xIsCreated THEN
	P_BV_2.Delete();
END_IF;

(* Q_BV_3 *)
IF Q_BV_3.xIsCreated THEN
	Q_BV_3.Delete();
END_IF;

(* R_BV_4 *)
IF R_BV_4.xIsCreated THEN
	R_BV_4.Delete();
END_IF;

(* S_BV_5 *)
IF S_BV_5.xIsCreated THEN
	S_BV_5.Delete();
END_IF;
(* Delete Struct View *)
IF GVL_BACNET.fbBacNetParameter.proDestroyBacNetOverrideXmlNode THEN
	fcXMLDeleteOverrideNode(fcBacNetIdToIdWitType(TO_DINT(CONCAT(TO_STRING(OBJ_ID_BASE),'1')),WagoTypesBacNet.eBACnetObjectType.BACnet_structured_view));
	fcXMLDeleteStructuredViewFromDevice(fcBacNetIdToIdWitType(TO_DINT(CONCAT(TO_STRING(OBJ_ID_BASE),'1')),WagoTypesBacNet.eBACnetObjectType.BACnet_structured_view));
END_IF;
metDELETE := 	A_DV_1.xIsCreated OR 
				B_CL_1.xIsCreated OR
				C_CL_2.xIsCreated OR				
				E_CL_4.xIsCreated OR
				F_EL_1.xIsCreated OR
				G_NC_1.xIsCreated OR
				G_NC_2.xIsCreated OR
				G_NC_3.xIsCreated OR
				G_NC_4.xIsCreated OR
				H_NC_32.xIsCreated OR
				H_NC_33.xIsCreated OR
				H_NC_34.xIsCreated OR
				H_NC_35.xIsCreated OR
				I_NC_64.xIsCreated OR
				I_NC_65.xIsCreated OR
				I_NC_66.xIsCreated OR
				I_NC_67.xIsCreated OR
				J_NC_96.xIsCreated OR
				J_NC_97.xIsCreated OR
				J_NC_98.xIsCreated OR
				J_NC_99.xIsCreated OR
				K_NC_128.xIsCreated OR
				K_NC_129.xIsCreated OR
				K_NC_130.xIsCreated OR
				K_NC_131.xIsCreated OR
				L_NC_160.xIsCreated OR
				L_NC_161.xIsCreated OR
				L_NC_162.xIsCreated OR
				L_NC_163.xIsCreated OR
				M_NC_192.xIsCreated OR
				M_NC_193.xIsCreated OR
				N_NC_224.xIsCreated OR
				N_NC_225.xIsCreated OR
				O_BV_1.xIsCreated OR
				P_BV_2.xIsCreated OR
				Q_BV_3.xIsCreated OR
				R_BV_4.xIsCreated OR
				S_BV_5.xIsCreated ;
(* Reset Create Case *)
usiCreateCase := 1;
END_METHOD

METHOD metCREATE_KBOB_2017_V1 : BOOL;
VAR_INPUT
END_VAR
VAR
	oStatus		:	WagoSysErrorBase.FbResult;
	usiErrors	:	USINT;
END_VAR
(* Resett *)
usiErrors := 0;	

(* Create Objeccts *)
CASE usiCreateCase OF
	1:	
		usiErrors := usiErrors + TO_USINT(NOT metCreate_A_DV_1());
	2:
		usiErrors := usiErrors + TO_USINT(NOT metCreate_B_CL_1());
	3:	
		usiErrors := usiErrors + TO_USINT(NOT metCreate_C_CL_2());
	4:	
		usiErrors := usiErrors + TO_USINT(NOT metCreate_D_CL_3());
	5:
		usiErrors := usiErrors + TO_USINT(NOT metCreate_E_CL_4());
	6:	
		usiErrors := usiErrors + TO_USINT(NOT metCreate_F_EL_1());
	7:
		usiErrors := usiErrors + TO_USINT(NOT metCreate_G_NC_1());
	8:	
		usiErrors := usiErrors + TO_USINT(NOT metCreate_G_NC_2());
	9:
		usiErrors := usiErrors + TO_USINT(NOT metCreate_G_NC_3());
	10:
		usiErrors := usiErrors + TO_USINT(NOT metCreate_G_NC_4());
	11:	
		usiErrors := usiErrors + TO_USINT(NOT metCreate_H_NC_32());
	12:
		usiErrors := usiErrors + TO_USINT(NOT metCreate_H_NC_33());
	13:
		usiErrors := usiErrors + TO_USINT(NOT metCreate_H_NC_34());
	14:
		usiErrors := usiErrors + TO_USINT(NOT metCreate_H_NC_35());
	15:
		usiErrors := usiErrors + TO_USINT(NOT metCreate_I_NC_64());
	16:
		usiErrors := usiErrors + TO_USINT(NOT metCreate_I_NC_65());
	17:
		usiErrors := usiErrors + TO_USINT(NOT metCreate_I_NC_66());
	18:
		usiErrors := usiErrors + TO_USINT(NOT metCreate_I_NC_67());
	19:
		usiErrors := usiErrors + TO_USINT(NOT metCreate_J_NC_96());
	20:
		usiErrors := usiErrors + TO_USINT(NOT metCreate_J_NC_97());
	21:
		usiErrors := usiErrors + TO_USINT(NOT metCreate_J_NC_98());
	22:
		usiErrors := usiErrors + TO_USINT(NOT metCreate_J_NC_99());
	23:
		usiErrors := usiErrors + TO_USINT(NOT metCreate_K_NC_128());
	24:
		usiErrors := usiErrors + TO_USINT(NOT metCreate_K_NC_129());
	25:
		usiErrors := usiErrors + TO_USINT(NOT metCreate_K_NC_130());
	26:
		usiErrors := usiErrors + TO_USINT(NOT metCreate_K_NC_131());
	27:
		usiErrors := usiErrors + TO_USINT(NOT metCreate_L_NC_160());
	28:
		usiErrors := usiErrors + TO_USINT(NOT metCreate_L_NC_161());
	29:
		usiErrors := usiErrors + TO_USINT(NOT metCreate_L_NC_162());
	30:
		usiErrors := usiErrors + TO_USINT(NOT metCreate_L_NC_163());
	31:
		usiErrors := usiErrors + TO_USINT(NOT metCreate_M_NC_192());
	32:
		usiErrors := usiErrors + TO_USINT(NOT metCreate_M_NC_193());
	33:
		usiErrors := usiErrors + TO_USINT(NOT metCreate_N_NC_224());
	34:
		usiErrors := usiErrors + TO_USINT(NOT metCreate_N_NC_225());
	35:
		usiErrors := usiErrors + TO_USINT(NOT metCreate_O_BV_1());
	36:
		usiErrors := usiErrors + TO_USINT(NOT metCreate_P_BV_2());
	37:
		usiErrors := usiErrors + TO_USINT(NOT metCreate_Q_BV_3());
	38:
		usiErrors := usiErrors + TO_USINT(NOT metCreate_R_BV_4());
	39:
		usiErrors := usiErrors + TO_USINT(NOT metCreate_S_BV_5());
	0: 
		usiCreateCase := 1;
ELSE
	usiCreateCase := 0;
END_CASE;

(* STRUCT VIEW *)
metCREATE_STRUCTVIEW_KBOB_2017_V1();

(* OK = 0*)
metCREATE_KBOB_2017_V1 := NOT TO_BOOL(usiErrors);
END_METHOD

METHOD metCREATE_STRUCTVIEW_KBOB_2017_V1 : BOOL
VAR_INPUT
END_VAR
CASE usiCreateCase OF
	1:
		fcXMLStructuredView(THIS^,A_DV_1.IObjectIdentifier);			
	2:                                                                 
		fcXMLStructuredView(THIS^,B_CL_1.IObjectIdentifier);            
	3:                                                                 
		fcXMLStructuredView(THIS^,C_CL_2.IObjectIdentifier);            
	4:                                                                 
		fcXMLStructuredView(THIS^,D_CL_3.IObjectIdentifier);            
	5:                                                                 
		fcXMLStructuredView(THIS^,E_CL_4.IObjectIdentifier);            
	6:                                                                 
		fcXMLStructuredView(THIS^,F_EL_1.IObjectIdentifier);            
	7:                                                                 
		fcXMLStructuredView(THIS^,G_NC_1.IObjectIdentifier);            
	8:                                                                 
		fcXMLStructuredView(THIS^,G_NC_2.IObjectIdentifier);            
	9:                                                                 
		fcXMLStructuredView(THIS^,G_NC_3.IObjectIdentifier);            
	10:                                                                
		fcXMLStructuredView(THIS^,G_NC_4.IObjectIdentifier);            
	11:                                                                
		fcXMLStructuredView(THIS^,H_NC_32.IObjectIdentifier);           
	12:                                                                
		fcXMLStructuredView(THIS^,H_NC_33.IObjectIdentifier);  
	13:                                                                
		fcXMLStructuredView(THIS^,H_NC_34.IObjectIdentifier);  
	14:                                                                
		fcXMLStructuredView(THIS^,H_NC_35.IObjectIdentifier);           
	15:                                                                
		 fcXMLStructuredView(THIS^,I_NC_64.IObjectIdentifier);           
	16:                                                                
		 fcXMLStructuredView(THIS^,I_NC_65.IObjectIdentifier);           
	17:                                                                
		 fcXMLStructuredView(THIS^,I_NC_66.IObjectIdentifier);           
	18:	                                                               
		 fcXMLStructuredView(THIS^,I_NC_67.IObjectIdentifier);           
	19:                                                                
		 fcXMLStructuredView(THIS^,J_NC_96.IObjectIdentifier);           
	20:                                                                
		 fcXMLStructuredView(THIS^,J_NC_97.IObjectIdentifier);           
	21:                                                                
		 fcXMLStructuredView(THIS^,J_NC_98.IObjectIdentifier);           
	22:                                                                
		 fcXMLStructuredView(THIS^,J_NC_99.IObjectIdentifier);           
	23:                                                                
		 fcXMLStructuredView(THIS^,K_NC_128.IObjectIdentifier);          
	24:                                                                
		 fcXMLStructuredView(THIS^,K_NC_129.IObjectIdentifier);          
	25:                                                                
		 fcXMLStructuredView(THIS^,K_NC_130.IObjectIdentifier);          
	26:                                                                
		 fcXMLStructuredView(THIS^,K_NC_131.IObjectIdentifier);          
	27:                                                                
		 fcXMLStructuredView(THIS^,L_NC_160.IObjectIdentifier);          
	28:                                                                
		 fcXMLStructuredView(THIS^,L_NC_161.IObjectIdentifier);          
	29:                                                                
		 fcXMLStructuredView(THIS^,L_NC_162.IObjectIdentifier);          
	30:                                                                
		 fcXMLStructuredView(THIS^,L_NC_163.IObjectIdentifier);		    
	31:                                                                
		 fcXMLStructuredView(THIS^,M_NC_192.IObjectIdentifier);          
	32:                                                                
		 fcXMLStructuredView(THIS^,M_NC_193.IObjectIdentifier);          
	33:                                                                
		 fcXMLStructuredView(THIS^,N_NC_224.IObjectIdentifier);          
	34:                                                                
		 fcXMLStructuredView(THIS^,N_NC_225.IObjectIdentifier);	        
	35:                                                                
		 fcXMLStructuredView(THIS^,O_BV_1.IObjectIdentifier);            
	36:                                                                
		 fcXMLStructuredView(THIS^,P_BV_2.IObjectIdentifier);            
	37:                                                                
		fcXMLStructuredView(THIS^,Q_BV_3.IObjectIdentifier);            
	38:                                                                
		fcXMLStructuredView(THIS^,R_BV_4.IObjectIdentifier);            
	39:                                                                
		fcXMLStructuredView(THIS^,S_BV_5.IObjectIdentifier);            	                                                               
		fcXMLAddStructuredViewToDevice(THIS^);	                            
	0:                                                                 
		usiCreateCase := 1;                                             
ELSE
	usiCreateCase := 0;
END_CASE
END_METHOD

METHOD metCREATE_KBOB_2021_V2 : BOOL;
VAR_INPUT
END_VAR
VAR
	oStatus		:	WagoSysErrorBase.FbResult;
	usiErrors	:	USINT;
END_VAR
(* Resett *)
usiErrors := 0;	

(* Create Objeccts *)
CASE usiCreateCase OF
	1:	
		usiErrors := usiErrors + TO_USINT(NOT metCreate_A_DV_1());
	2:
		usiErrors := usiErrors + TO_USINT(NOT metCreate_B_CL_1());
	3:	
		usiErrors := usiErrors + TO_USINT(NOT metCreate_C_CL_2());
	4:	
		usiErrors := usiErrors + TO_USINT(NOT metCreate_D_CL_3());
	5:
		usiErrors := usiErrors + TO_USINT(NOT metCreate_E_CL_4());
	6:	
		usiErrors := usiErrors + TO_USINT(NOT metCreate_F_EL_1());
	7:
		usiErrors := usiErrors + TO_USINT(NOT metCreate_G_NC_1());
	8:	
		usiErrors := usiErrors + TO_USINT(NOT metCreate_G_NC_2());
	9:
		usiErrors := usiErrors + TO_USINT(NOT metCreate_G_NC_3());
	10:
		usiErrors := usiErrors + TO_USINT(NOT metCreate_G_NC_4());
	11:	
		usiErrors := usiErrors + TO_USINT(NOT metCreate_H_NC_32());
	12:
		usiErrors := usiErrors + TO_USINT(NOT metCreate_H_NC_33());
	13:
		usiErrors := usiErrors + TO_USINT(NOT metCreate_H_NC_34());
	14:
		usiErrors := usiErrors + TO_USINT(NOT metCreate_H_NC_35());
	15:
		usiErrors := usiErrors + TO_USINT(NOT metCreate_I_NC_64());
	16:
		usiErrors := usiErrors + TO_USINT(NOT metCreate_I_NC_65());
	17:
		usiErrors := usiErrors + TO_USINT(NOT metCreate_I_NC_66());
	18:
		usiErrors := usiErrors + TO_USINT(NOT metCreate_I_NC_67());
	19:
		usiErrors := usiErrors + TO_USINT(NOT metCreate_J_NC_96());
	20:
		usiErrors := usiErrors + TO_USINT(NOT metCreate_J_NC_97());
	21:
		usiErrors := usiErrors + TO_USINT(NOT metCreate_J_NC_98());
	22:
		usiErrors := usiErrors + TO_USINT(NOT metCreate_J_NC_99());
	23:
		usiErrors := usiErrors + TO_USINT(NOT metCreate_K_NC_128());
	24:
		usiErrors := usiErrors + TO_USINT(NOT metCreate_K_NC_129());
	25:
		usiErrors := usiErrors + TO_USINT(NOT metCreate_K_NC_130());
	26:
		usiErrors := usiErrors + TO_USINT(NOT metCreate_K_NC_131());
	27:
		usiErrors := usiErrors + TO_USINT(NOT metCreate_L_NC_160());
	28:
		usiErrors := usiErrors + TO_USINT(NOT metCreate_L_NC_161());
	29:
		usiErrors := usiErrors + TO_USINT(NOT metCreate_L_NC_162());
	30:
		usiErrors := usiErrors + TO_USINT(NOT metCreate_L_NC_163());
	31:
		usiErrors := usiErrors + TO_USINT(NOT metCreate_M_NC_192());
	32:
		usiErrors := usiErrors + TO_USINT(NOT metCreate_M_NC_193());
	33:
		usiErrors := usiErrors + TO_USINT(NOT metCreate_N_NC_224());
	34:
		usiErrors := usiErrors + TO_USINT(NOT metCreate_N_NC_225());
	35:
		usiErrors := usiErrors + TO_USINT(NOT metCreate_O_BV_1());
	36:
		usiErrors := usiErrors + TO_USINT(NOT metCreate_P_BV_2());
	37:
		usiErrors := usiErrors + TO_USINT(NOT metCreate_Q_BV_3());
	38:
		usiErrors := usiErrors + TO_USINT(NOT metCreate_R_BV_4());
	39:
		usiErrors := usiErrors + TO_USINT(NOT metCreate_S_BV_5());
	0: 
		usiCreateCase := 1;
ELSE
	usiCreateCase := 0;
END_CASE;

(* STRUCT VIEW *)
metCREATE_STRUCTVIEW_KBOB_2021_V2();

(* OK = 0*)
metCREATE_KBOB_2021_V2 := NOT TO_BOOL(usiErrors);
END_METHOD

METHOD metCREATE_STRUCTVIEW_KBOB_2021_V2 : BOOL
VAR_INPUT
END_VAR
CASE usiCreateCase OF
	1:
		fcXMLStructuredView(THIS^,A_DV_1.IObjectIdentifier);			
	2:                                                                 
		fcXMLStructuredView(THIS^,B_CL_1.IObjectIdentifier);            
	3:                                                                 
		fcXMLStructuredView(THIS^,C_CL_2.IObjectIdentifier);            
	4:                                                                 
		fcXMLStructuredView(THIS^,D_CL_3.IObjectIdentifier);            
	5:                                                                 
		fcXMLStructuredView(THIS^,E_CL_4.IObjectIdentifier);            
	6:                                                                 
		fcXMLStructuredView(THIS^,F_EL_1.IObjectIdentifier);            
	7:                                                                 
		fcXMLStructuredView(THIS^,G_NC_1.IObjectIdentifier);            
	8:                                                                 
		fcXMLStructuredView(THIS^,G_NC_2.IObjectIdentifier);            
	9:                                                                 
		fcXMLStructuredView(THIS^,G_NC_3.IObjectIdentifier);            
	10:                                                                
		fcXMLStructuredView(THIS^,G_NC_4.IObjectIdentifier);            
	11:                                                                
		fcXMLStructuredView(THIS^,H_NC_32.IObjectIdentifier);           
	12:                                                                
		fcXMLStructuredView(THIS^,H_NC_33.IObjectIdentifier);  
	13:                                                                
		fcXMLStructuredView(THIS^,H_NC_34.IObjectIdentifier);  
	14:                                                                
		fcXMLStructuredView(THIS^,H_NC_35.IObjectIdentifier);           
	15:                                                                
		 fcXMLStructuredView(THIS^,I_NC_64.IObjectIdentifier);           
	16:                                                                
		 fcXMLStructuredView(THIS^,I_NC_65.IObjectIdentifier);           
	17:                                                                
		 fcXMLStructuredView(THIS^,I_NC_66.IObjectIdentifier);           
	18:	                                                               
		 fcXMLStructuredView(THIS^,I_NC_67.IObjectIdentifier);           
	19:                                                                
		 fcXMLStructuredView(THIS^,J_NC_96.IObjectIdentifier);           
	20:                                                                
		 fcXMLStructuredView(THIS^,J_NC_97.IObjectIdentifier);           
	21:                                                                
		 fcXMLStructuredView(THIS^,J_NC_98.IObjectIdentifier);           
	22:                                                                
		 fcXMLStructuredView(THIS^,J_NC_99.IObjectIdentifier);           
	23:                                                                
		 fcXMLStructuredView(THIS^,K_NC_128.IObjectIdentifier);          
	24:                                                                
		 fcXMLStructuredView(THIS^,K_NC_129.IObjectIdentifier);          
	25:                                                                
		 fcXMLStructuredView(THIS^,K_NC_130.IObjectIdentifier);          
	26:                                                                
		 fcXMLStructuredView(THIS^,K_NC_131.IObjectIdentifier);          
	27:                                                                
		 fcXMLStructuredView(THIS^,L_NC_160.IObjectIdentifier);          
	28:                                                                
		 fcXMLStructuredView(THIS^,L_NC_161.IObjectIdentifier);          
	29:                                                                
		 fcXMLStructuredView(THIS^,L_NC_162.IObjectIdentifier);          
	30:                                                                
		 fcXMLStructuredView(THIS^,L_NC_163.IObjectIdentifier);		    
	31:                                                                
		 fcXMLStructuredView(THIS^,M_NC_192.IObjectIdentifier);          
	32:                                                                
		 fcXMLStructuredView(THIS^,M_NC_193.IObjectIdentifier);          
	33:                                                                
		 fcXMLStructuredView(THIS^,N_NC_224.IObjectIdentifier);          
	34:                                                                
		 fcXMLStructuredView(THIS^,N_NC_225.IObjectIdentifier);	        
	35:                                                                
		 fcXMLStructuredView(THIS^,O_BV_1.IObjectIdentifier);            
	36:                                                                
		 fcXMLStructuredView(THIS^,P_BV_2.IObjectIdentifier);            
	37:                                                                
		fcXMLStructuredView(THIS^,Q_BV_3.IObjectIdentifier);            
	38:                                                                
		fcXMLStructuredView(THIS^,R_BV_4.IObjectIdentifier);            
	39:                                                                
		fcXMLStructuredView(THIS^,S_BV_5.IObjectIdentifier);            	                                                               
		fcXMLAddStructuredViewToDevice(THIS^);	                            
	0:                                                                 
		usiCreateCase := 1;                                             
ELSE
	usiCreateCase := 0;
END_CASE
END_METHOD

METHOD metCREATE : BOOL;
VAR_INPUT
END_VAR
VAR
	oStatus		:	WagoSysErrorBase.FbResult;
	usiErrors	:	USINT;
END_VAR
(* Get Revision *)
CASE GVL_BACNET.fbBacNetParameter.proKBOB_REV OF
	(* KBOB 2021 V2 *)
	enKBOB_REV.KBOB_REV2021_V2:
		usiErrors := usiErrors + TO_USINT(NOT metCREATE_KBOB_2021_V2());
	(* KBOB 2017 V1 *)
	enKBOB_REV.KBOB_REV2017_V1:
		usiErrors := usiErrors + TO_USINT(NOT metCREATE_KBOB_2017_V1());
	(* Default *)
	ELSE
		usiErrors := usiErrors + TO_USINT(NOT metCREATE_KBOB_2021_V2());
END_CASE;

(* OK = 0*)
xErrorCreate := TO_BOOL(usiErrors);
metCREATE := NOT TO_BOOL(usiErrors) AND usiCreateCase = usiAnzBacNetObj;
END_METHOD

METHOD metCreate_L_NC_160 : BOOL

VAR

END_VAR
(* L_NC_160*)
IF NOT L_NC_160.xIsCreated THEN
	(* Ziel						UTF8->ASCII						OBJ_NAME_BASE			BacNet Text		Textlistname									BacNet Funktion																	BacNet Textlist type												TextId		*)
	L_NC_160._sObjectName		:=	fcUtfToAscii(Standard.CONCAT(	OBJ_NAME_BASE		,	fcGetBcText(	GVL_BACNET.fbBacNetParameter.metGetTextListName(enTypeOfBacNetFunktionIn := enTypeOfBacNetFunktion.Type_Automationsstation,		enTypeOfBacNetTextListIn := enTypeOfBacNetTextList.ENDING		),	'L_NC_160')));
	L_NC_160._sDescription	:= 	fcUtfToAscii(Standard.CONCAT(	OBJ_NAME_DESCRIPTION,	fcGetBcText(	GVL_BACNET.fbBacNetParameter.metGetTextListName(enTypeOfBacNetFunktionIn := enTypeOfBacNetFunktion.Type_Automationsstation,		enTypeOfBacNetTextListIn := enTypeOfBacNetTextList.DESCRIPTION	),	'L_NC_160')));
	(* Create Id from Base Id and Object Nr (Last nummber of Name *)	
	L_NC_160.Create(diInstance := 160);
	(* Check if Created *)
	IF L_NC_160.xIsCreated THEN
		(* Set Group *)
		L_NC_160.setPropertyGroup(WagoTypesBacNet.eBACnetPropertyIdentifier.PROP_DESCRIPTION							,WagoTypesBacNet.eBACnetPropertyUpdateGroup.GROUP_CYCLIC);
		
		(* Set Ack Req *)
		L_NC_160.IAckRequired.xToOffNormal	:= FALSE;
		L_NC_160.IAckRequired.xToFault		:= FALSE;
		L_NC_160.IAckRequired.xToNormal		:= FALSE;
		
		(* Ziel												UTF8->ASCII		BacNet Text		Textlistname									BacNet Funktion																	BacNet Textlist type												TextId		*)
		L_NC_160.IEventMessageTextsConfig.sToOffNormal	:=	fcUtfToAscii(	fcGetBcText(	GVL_BACNET.fbBacNetParameter.metGetTextListName(enTypeOfBacNetFunktionIn := enTypeOfBacNetFunktion.Type_Automationsstation,		enTypeOfBacNetTextListIn := enTypeOfBacNetTextList.EVENTMESSAGE	),	'L_NC_160_ToOffNormal'	));		
		L_NC_160.IEventMessageTextsConfig.sToFault		:=	fcUtfToAscii(	fcGetBcText(	GVL_BACNET.fbBacNetParameter.metGetTextListName(enTypeOfBacNetFunktionIn := enTypeOfBacNetFunktion.Type_Automationsstation,		enTypeOfBacNetTextListIn := enTypeOfBacNetTextList.EVENTMESSAGE	),	'L_NC_160_ToFault'		));		
		L_NC_160.IEventMessageTextsConfig.sToNormal		:=	fcUtfToAscii(	fcGetBcText(	GVL_BACNET.fbBacNetParameter.metGetTextListName(enTypeOfBacNetFunktionIn := enTypeOfBacNetFunktion.Type_Automationsstation,		enTypeOfBacNetTextListIn := enTypeOfBacNetTextList.EVENTMESSAGE	),	'L_NC_160_ToNormal'		));		
		
		(* Notification Class & Type *)
		L_NC_160.udiNotificationClass					:=  160;	
		L_NC_160.eNotifyType							:= 	WagoTypesBACnet.eBACnetNotifyType.NOTIFY_TYPE_ALARM;
		(* Ziel												Convert			BacNet Text		Textlistname									BacNet Funktion																	BacNet Textlist type												TextId		*)	
		L_NC_160.IPriority.usiToOffNormal				:= 	TO_USINT(fcUtfToAscii(	fcGetBcText(	GVL_BACNET.fbBacNetParameter.metGetTextListName(enTypeOfBacNetFunktionIn := enTypeOfBacNetFunktion.Type_Automationsstation,		enTypeOfBacNetTextListIn := enTypeOfBacNetTextList.NC	),	'L_NC_160_Prio_ToOffNormal'	)));	
		L_NC_160.IPriority.usiToFault					:= 	TO_USINT(fcUtfToAscii(	fcGetBcText(	GVL_BACNET.fbBacNetParameter.metGetTextListName(enTypeOfBacNetFunktionIn := enTypeOfBacNetFunktion.Type_Automationsstation,		enTypeOfBacNetTextListIn := enTypeOfBacNetTextList.NC	),	'L_NC_160_Prio_ToFault'		)));	
		L_NC_160.IPriority.usiToNormal					:= 	TO_USINT(fcUtfToAscii(	fcGetBcText(	GVL_BACNET.fbBacNetParameter.metGetTextListName(enTypeOfBacNetFunktionIn := enTypeOfBacNetFunktion.Type_Automationsstation,		enTypeOfBacNetTextListIn := enTypeOfBacNetTextList.NC	),	'L_NC_160_Prio_ToNormal'		)));	
		
	ELSE
		L_NC_160.Delete();
	END_IF;
	(* Get Status *)
	metCreate_L_NC_160 := L_NC_160.xIsCreated;	
END_IF;
END_METHOD

METHOD metCreate_L_NC_161 : BOOL

VAR

END_VAR
(* L_NC_161*)
IF NOT L_NC_161.xIsCreated THEN
	(* Ziel						UTF8->ASCII						OBJ_NAME_BASE			BacNet Text		Textlistname									BacNet Funktion																	BacNet Textlist type												TextId		*)
	L_NC_161._sObjectName		:=	fcUtfToAscii(Standard.CONCAT(	OBJ_NAME_BASE		,	fcGetBcText(	GVL_BACNET.fbBacNetParameter.metGetTextListName(enTypeOfBacNetFunktionIn := enTypeOfBacNetFunktion.Type_Automationsstation,		enTypeOfBacNetTextListIn := enTypeOfBacNetTextList.ENDING		),	'L_NC_161')));
	L_NC_161._sDescription	:= 	fcUtfToAscii(Standard.CONCAT(	OBJ_NAME_DESCRIPTION,	fcGetBcText(	GVL_BACNET.fbBacNetParameter.metGetTextListName(enTypeOfBacNetFunktionIn := enTypeOfBacNetFunktion.Type_Automationsstation,		enTypeOfBacNetTextListIn := enTypeOfBacNetTextList.DESCRIPTION	),	'L_NC_161')));
	(* Create Id from Base Id and Object Nr (Last nummber of Name *)	
	L_NC_161.Create(diInstance := 161);
	(* Check if Created *)
	IF L_NC_161.xIsCreated THEN
		(* Set Group *)
		L_NC_161.setPropertyGroup(WagoTypesBacNet.eBACnetPropertyIdentifier.PROP_DESCRIPTION							,WagoTypesBacNet.eBACnetPropertyUpdateGroup.GROUP_CYCLIC);
		
		(* Set Ack Req *)
		L_NC_161.IAckRequired.xToOffNormal	:= FALSE;
		L_NC_161.IAckRequired.xToFault		:= TRUE;
		L_NC_161.IAckRequired.xToNormal		:= FALSE;
		
		(* Ziel												UTF8->ASCII		BacNet Text		Textlistname									BacNet Funktion																	BacNet Textlist type												TextId		*)
		L_NC_161.IEventMessageTextsConfig.sToOffNormal	:=	fcUtfToAscii(	fcGetBcText(	GVL_BACNET.fbBacNetParameter.metGetTextListName(enTypeOfBacNetFunktionIn := enTypeOfBacNetFunktion.Type_Automationsstation,		enTypeOfBacNetTextListIn := enTypeOfBacNetTextList.EVENTMESSAGE	),	'L_NC_161_ToOffNormal'	));		
		L_NC_161.IEventMessageTextsConfig.sToFault		:=	fcUtfToAscii(	fcGetBcText(	GVL_BACNET.fbBacNetParameter.metGetTextListName(enTypeOfBacNetFunktionIn := enTypeOfBacNetFunktion.Type_Automationsstation,		enTypeOfBacNetTextListIn := enTypeOfBacNetTextList.EVENTMESSAGE	),	'L_NC_161_ToFault'		));		
		L_NC_161.IEventMessageTextsConfig.sToNormal		:=	fcUtfToAscii(	fcGetBcText(	GVL_BACNET.fbBacNetParameter.metGetTextListName(enTypeOfBacNetFunktionIn := enTypeOfBacNetFunktion.Type_Automationsstation,		enTypeOfBacNetTextListIn := enTypeOfBacNetTextList.EVENTMESSAGE	),	'L_NC_161_ToNormal'		));		
		
		(* Notification Class & Type *)
		L_NC_161.udiNotificationClass					:=  161;	
		L_NC_161.eNotifyType							:= 	WagoTypesBACnet.eBACnetNotifyType.NOTIFY_TYPE_ALARM;
		(* Ziel												Convert			BacNet Text		Textlistname									BacNet Funktion																	BacNet Textlist type												TextId		*)	
		L_NC_161.IPriority.usiToOffNormal				:= 	TO_USINT(fcUtfToAscii(	fcGetBcText(	GVL_BACNET.fbBacNetParameter.metGetTextListName(enTypeOfBacNetFunktionIn := enTypeOfBacNetFunktion.Type_Automationsstation,		enTypeOfBacNetTextListIn := enTypeOfBacNetTextList.NC	),	'L_NC_161_Prio_ToOffNormal'	)));	
		L_NC_161.IPriority.usiToFault					:= 	TO_USINT(fcUtfToAscii(	fcGetBcText(	GVL_BACNET.fbBacNetParameter.metGetTextListName(enTypeOfBacNetFunktionIn := enTypeOfBacNetFunktion.Type_Automationsstation,		enTypeOfBacNetTextListIn := enTypeOfBacNetTextList.NC	),	'L_NC_161_Prio_ToFault'		)));	
		L_NC_161.IPriority.usiToNormal					:= 	TO_USINT(fcUtfToAscii(	fcGetBcText(	GVL_BACNET.fbBacNetParameter.metGetTextListName(enTypeOfBacNetFunktionIn := enTypeOfBacNetFunktion.Type_Automationsstation,		enTypeOfBacNetTextListIn := enTypeOfBacNetTextList.NC	),	'L_NC_161_Prio_ToNormal'		)));	
		
	ELSE
		L_NC_161.Delete();
	END_IF;
	(* Get Status *)
	metCreate_L_NC_161 := L_NC_161.xIsCreated;	
END_IF;
END_METHOD

METHOD metCreate_L_NC_162 : BOOL

VAR

END_VAR
(* L_NC_162*)
IF NOT L_NC_162.xIsCreated THEN
	(* Ziel						UTF8->ASCII						OBJ_NAME_BASE			BacNet Text		Textlistname									BacNet Funktion																	BacNet Textlist type												TextId		*)
	L_NC_162._sObjectName		:=	fcUtfToAscii(Standard.CONCAT(	OBJ_NAME_BASE		,	fcGetBcText(	GVL_BACNET.fbBacNetParameter.metGetTextListName(enTypeOfBacNetFunktionIn := enTypeOfBacNetFunktion.Type_Automationsstation,		enTypeOfBacNetTextListIn := enTypeOfBacNetTextList.ENDING		),	'L_NC_162')));
	L_NC_162._sDescription	:= 	fcUtfToAscii(Standard.CONCAT(	OBJ_NAME_DESCRIPTION,	fcGetBcText(	GVL_BACNET.fbBacNetParameter.metGetTextListName(enTypeOfBacNetFunktionIn := enTypeOfBacNetFunktion.Type_Automationsstation,		enTypeOfBacNetTextListIn := enTypeOfBacNetTextList.DESCRIPTION	),	'L_NC_162')));
	(* Create Id from Base Id and Object Nr (Last nummber of Name *)	
	L_NC_162.Create(diInstance := 162);
	(* Check if Created *)
	IF L_NC_162.xIsCreated THEN
		(* Set Group *)
		L_NC_162.setPropertyGroup(WagoTypesBacNet.eBACnetPropertyIdentifier.PROP_DESCRIPTION							,WagoTypesBacNet.eBACnetPropertyUpdateGroup.GROUP_CYCLIC);
		
		(* Set Ack Req *)
		L_NC_162.IAckRequired.xToOffNormal	:= TRUE;
		L_NC_162.IAckRequired.xToFault		:= TRUE;
		L_NC_162.IAckRequired.xToNormal		:= FALSE;
		
		(* Ziel												UTF8->ASCII		BacNet Text		Textlistname									BacNet Funktion																	BacNet Textlist type												TextId		*)
		L_NC_162.IEventMessageTextsConfig.sToOffNormal	:=	fcUtfToAscii(	fcGetBcText(	GVL_BACNET.fbBacNetParameter.metGetTextListName(enTypeOfBacNetFunktionIn := enTypeOfBacNetFunktion.Type_Automationsstation,		enTypeOfBacNetTextListIn := enTypeOfBacNetTextList.EVENTMESSAGE	),	'L_NC_162_ToOffNormal'	));		
		L_NC_162.IEventMessageTextsConfig.sToFault		:=	fcUtfToAscii(	fcGetBcText(	GVL_BACNET.fbBacNetParameter.metGetTextListName(enTypeOfBacNetFunktionIn := enTypeOfBacNetFunktion.Type_Automationsstation,		enTypeOfBacNetTextListIn := enTypeOfBacNetTextList.EVENTMESSAGE	),	'L_NC_162_ToFault'		));		
		L_NC_162.IEventMessageTextsConfig.sToNormal		:=	fcUtfToAscii(	fcGetBcText(	GVL_BACNET.fbBacNetParameter.metGetTextListName(enTypeOfBacNetFunktionIn := enTypeOfBacNetFunktion.Type_Automationsstation,		enTypeOfBacNetTextListIn := enTypeOfBacNetTextList.EVENTMESSAGE	),	'L_NC_162_ToNormal'		));		
		
		(* Notification Class & Type *)
		L_NC_162.udiNotificationClass					:=  162;	
		L_NC_162.eNotifyType							:= 	WagoTypesBACnet.eBACnetNotifyType.NOTIFY_TYPE_ALARM;
		(* Ziel												Convert			BacNet Text		Textlistname									BacNet Funktion																	BacNet Textlist type												TextId		*)	
		L_NC_162.IPriority.usiToOffNormal				:= 	TO_USINT(fcUtfToAscii(	fcGetBcText(	GVL_BACNET.fbBacNetParameter.metGetTextListName(enTypeOfBacNetFunktionIn := enTypeOfBacNetFunktion.Type_Automationsstation,		enTypeOfBacNetTextListIn := enTypeOfBacNetTextList.NC	),	'L_NC_162_Prio_ToOffNormal'	)));	
		L_NC_162.IPriority.usiToFault					:= 	TO_USINT(fcUtfToAscii(	fcGetBcText(	GVL_BACNET.fbBacNetParameter.metGetTextListName(enTypeOfBacNetFunktionIn := enTypeOfBacNetFunktion.Type_Automationsstation,		enTypeOfBacNetTextListIn := enTypeOfBacNetTextList.NC	),	'L_NC_162_Prio_ToFault'		)));	
		L_NC_162.IPriority.usiToNormal					:= 	TO_USINT(fcUtfToAscii(	fcGetBcText(	GVL_BACNET.fbBacNetParameter.metGetTextListName(enTypeOfBacNetFunktionIn := enTypeOfBacNetFunktion.Type_Automationsstation,		enTypeOfBacNetTextListIn := enTypeOfBacNetTextList.NC	),	'L_NC_162_Prio_ToNormal'		)));	
		
	ELSE
		L_NC_162.Delete();
	END_IF;
	(* Get Status *)
	metCreate_L_NC_162 := L_NC_162.xIsCreated;	
END_IF;
END_METHOD

METHOD metCreate_L_NC_163 : BOOL

VAR

END_VAR
(* L_NC_163*)
IF NOT L_NC_163.xIsCreated THEN
	(* Ziel						UTF8->ASCII						OBJ_NAME_BASE			BacNet Text		Textlistname									BacNet Funktion																	BacNet Textlist type												TextId		*)
	L_NC_163._sObjectName		:=	fcUtfToAscii(Standard.CONCAT(	OBJ_NAME_BASE		,	fcGetBcText(	GVL_BACNET.fbBacNetParameter.metGetTextListName(enTypeOfBacNetFunktionIn := enTypeOfBacNetFunktion.Type_Automationsstation,		enTypeOfBacNetTextListIn := enTypeOfBacNetTextList.ENDING		),	'L_NC_163')));
	L_NC_163._sDescription	:= 	fcUtfToAscii(Standard.CONCAT(	OBJ_NAME_DESCRIPTION,	fcGetBcText(	GVL_BACNET.fbBacNetParameter.metGetTextListName(enTypeOfBacNetFunktionIn := enTypeOfBacNetFunktion.Type_Automationsstation,		enTypeOfBacNetTextListIn := enTypeOfBacNetTextList.DESCRIPTION	),	'L_NC_163')));
	(* Create Id from Base Id and Object Nr (Last nummber of Name *)	
	L_NC_163.Create(diInstance := 163);
	(* Check if Created *)
	IF L_NC_163.xIsCreated THEN
		(* Set Group *)
		L_NC_163.setPropertyGroup(WagoTypesBacNet.eBACnetPropertyIdentifier.PROP_DESCRIPTION							,WagoTypesBacNet.eBACnetPropertyUpdateGroup.GROUP_CYCLIC);
		
		(* Set Ack Req *)
		L_NC_163.IAckRequired.xToOffNormal	:= TRUE;
		L_NC_163.IAckRequired.xToFault		:= TRUE;
		L_NC_163.IAckRequired.xToNormal		:= TRUE;
		
		(* Ziel												UTF8->ASCII		BacNet Text		Textlistname									BacNet Funktion																	BacNet Textlist type												TextId		*)
		L_NC_163.IEventMessageTextsConfig.sToOffNormal	:=	fcUtfToAscii(	fcGetBcText(	GVL_BACNET.fbBacNetParameter.metGetTextListName(enTypeOfBacNetFunktionIn := enTypeOfBacNetFunktion.Type_Automationsstation,		enTypeOfBacNetTextListIn := enTypeOfBacNetTextList.EVENTMESSAGE	),	'L_NC_163_ToOffNormal'	));		
		L_NC_163.IEventMessageTextsConfig.sToFault		:=	fcUtfToAscii(	fcGetBcText(	GVL_BACNET.fbBacNetParameter.metGetTextListName(enTypeOfBacNetFunktionIn := enTypeOfBacNetFunktion.Type_Automationsstation,		enTypeOfBacNetTextListIn := enTypeOfBacNetTextList.EVENTMESSAGE	),	'L_NC_163_ToFault'		));		
		L_NC_163.IEventMessageTextsConfig.sToNormal		:=	fcUtfToAscii(	fcGetBcText(	GVL_BACNET.fbBacNetParameter.metGetTextListName(enTypeOfBacNetFunktionIn := enTypeOfBacNetFunktion.Type_Automationsstation,		enTypeOfBacNetTextListIn := enTypeOfBacNetTextList.EVENTMESSAGE	),	'L_NC_163_ToNormal'		));		
		
		(* Notification Class & Type *)
		L_NC_163.udiNotificationClass					:=  163;	
		L_NC_163.eNotifyType							:= 	WagoTypesBACnet.eBACnetNotifyType.NOTIFY_TYPE_ALARM;
		(* Ziel												Convert			BacNet Text		Textlistname									BacNet Funktion																	BacNet Textlist type												TextId		*)	
		L_NC_163.IPriority.usiToOffNormal				:= 	TO_USINT(fcUtfToAscii(	fcGetBcText(	GVL_BACNET.fbBacNetParameter.metGetTextListName(enTypeOfBacNetFunktionIn := enTypeOfBacNetFunktion.Type_Automationsstation,		enTypeOfBacNetTextListIn := enTypeOfBacNetTextList.NC	),	'L_NC_163_Prio_ToOffNormal'	)));	
		L_NC_163.IPriority.usiToFault					:= 	TO_USINT(fcUtfToAscii(	fcGetBcText(	GVL_BACNET.fbBacNetParameter.metGetTextListName(enTypeOfBacNetFunktionIn := enTypeOfBacNetFunktion.Type_Automationsstation,		enTypeOfBacNetTextListIn := enTypeOfBacNetTextList.NC	),	'L_NC_163_Prio_ToFault'		)));	
		L_NC_163.IPriority.usiToNormal					:= 	TO_USINT(fcUtfToAscii(	fcGetBcText(	GVL_BACNET.fbBacNetParameter.metGetTextListName(enTypeOfBacNetFunktionIn := enTypeOfBacNetFunktion.Type_Automationsstation,		enTypeOfBacNetTextListIn := enTypeOfBacNetTextList.NC	),	'L_NC_163_Prio_ToNormal'		)));	
		
	ELSE
		L_NC_163.Delete();
	END_IF;
	(* Get Status *)
	metCreate_L_NC_163 := L_NC_163.xIsCreated;	
END_IF;
END_METHOD

METHOD metCreate_M_NC_192 : BOOL

VAR

END_VAR
(* M_NC_192*)
IF NOT M_NC_192.xIsCreated THEN
	(* Ziel						UTF8->ASCII						OBJ_NAME_BASE			BacNet Text		Textlistname									BacNet Funktion																	BacNet Textlist type												TextId		*)
	M_NC_192._sObjectName		:=	fcUtfToAscii(Standard.CONCAT(	OBJ_NAME_BASE		,	fcGetBcText(	GVL_BACNET.fbBacNetParameter.metGetTextListName(enTypeOfBacNetFunktionIn := enTypeOfBacNetFunktion.Type_Automationsstation,		enTypeOfBacNetTextListIn := enTypeOfBacNetTextList.ENDING		),	'M_NC_192')));
	M_NC_192._sDescription	:= 	fcUtfToAscii(Standard.CONCAT(	OBJ_NAME_DESCRIPTION,	fcGetBcText(	GVL_BACNET.fbBacNetParameter.metGetTextListName(enTypeOfBacNetFunktionIn := enTypeOfBacNetFunktion.Type_Automationsstation,		enTypeOfBacNetTextListIn := enTypeOfBacNetTextList.DESCRIPTION	),	'M_NC_192')));
	(* Create Id from Base Id and Object Nr (Last nummber of Name *)	
	M_NC_192.Create(diInstance := 192);
	(* Check if Created *)
	IF M_NC_192.xIsCreated THEN
		(* Set Group *)
		M_NC_192.setPropertyGroup(WagoTypesBacNet.eBACnetPropertyIdentifier.PROP_DESCRIPTION							,WagoTypesBacNet.eBACnetPropertyUpdateGroup.GROUP_CYCLIC);
		
		(* Set Ack Req *)
		M_NC_192.IAckRequired.xToOffNormal	:= FALSE;
		M_NC_192.IAckRequired.xToFault		:= FALSE;
		M_NC_192.IAckRequired.xToNormal		:= FALSE;
		
		(* Ziel												UTF8->ASCII		BacNet Text		Textlistname									BacNet Funktion																	BacNet Textlist type												TextId		*)
		M_NC_192.IEventMessageTextsConfig.sToOffNormal	:=	fcUtfToAscii(	fcGetBcText(	GVL_BACNET.fbBacNetParameter.metGetTextListName(enTypeOfBacNetFunktionIn := enTypeOfBacNetFunktion.Type_Automationsstation,		enTypeOfBacNetTextListIn := enTypeOfBacNetTextList.EVENTMESSAGE	),	'M_NC_192_ToOffNormal'	));		
		M_NC_192.IEventMessageTextsConfig.sToFault		:=	fcUtfToAscii(	fcGetBcText(	GVL_BACNET.fbBacNetParameter.metGetTextListName(enTypeOfBacNetFunktionIn := enTypeOfBacNetFunktion.Type_Automationsstation,		enTypeOfBacNetTextListIn := enTypeOfBacNetTextList.EVENTMESSAGE	),	'M_NC_192_ToFault'		));		
		M_NC_192.IEventMessageTextsConfig.sToNormal		:=	fcUtfToAscii(	fcGetBcText(	GVL_BACNET.fbBacNetParameter.metGetTextListName(enTypeOfBacNetFunktionIn := enTypeOfBacNetFunktion.Type_Automationsstation,		enTypeOfBacNetTextListIn := enTypeOfBacNetTextList.EVENTMESSAGE	),	'M_NC_192_ToNormal'		));		
		
		(* Notification Class & Type *)
		M_NC_192.udiNotificationClass					:=  192;	
		M_NC_192.eNotifyType							:= 	WagoTypesBACnet.eBACnetNotifyType.NOTIFY_TYPE_EVENT;
		(* Ziel												Convert			BacNet Text		Textlistname									BacNet Funktion																	BacNet Textlist type												TextId		*)	
		M_NC_192.IPriority.usiToOffNormal				:= 	TO_USINT(fcUtfToAscii(	fcGetBcText(	GVL_BACNET.fbBacNetParameter.metGetTextListName(enTypeOfBacNetFunktionIn := enTypeOfBacNetFunktion.Type_Automationsstation,		enTypeOfBacNetTextListIn := enTypeOfBacNetTextList.NC	),	'M_NC_192_Prio_ToOffNormal'	)));	
		M_NC_192.IPriority.usiToFault					:= 	TO_USINT(fcUtfToAscii(	fcGetBcText(	GVL_BACNET.fbBacNetParameter.metGetTextListName(enTypeOfBacNetFunktionIn := enTypeOfBacNetFunktion.Type_Automationsstation,		enTypeOfBacNetTextListIn := enTypeOfBacNetTextList.NC	),	'M_NC_192_Prio_ToFault'		)));	
		M_NC_192.IPriority.usiToNormal					:= 	TO_USINT(fcUtfToAscii(	fcGetBcText(	GVL_BACNET.fbBacNetParameter.metGetTextListName(enTypeOfBacNetFunktionIn := enTypeOfBacNetFunktion.Type_Automationsstation,		enTypeOfBacNetTextListIn := enTypeOfBacNetTextList.NC	),	'M_NC_192_Prio_ToNormal'		)));	
		
	ELSE
		M_NC_192.Delete();
	END_IF;
	(* Get Status *)
	metCreate_M_NC_192 := M_NC_192.xIsCreated;	
END_IF;
END_METHOD

METHOD metCreate_M_NC_193 : BOOL

VAR

END_VAR
(* M_NC_193*)
IF NOT M_NC_193.xIsCreated THEN
	(* Ziel						UTF8->ASCII						OBJ_NAME_BASE			BacNet Text		Textlistname									BacNet Funktion																	BacNet Textlist type												TextId		*)
	M_NC_193._sObjectName		:=	fcUtfToAscii(Standard.CONCAT(	OBJ_NAME_BASE		,	fcGetBcText(	GVL_BACNET.fbBacNetParameter.metGetTextListName(enTypeOfBacNetFunktionIn := enTypeOfBacNetFunktion.Type_Automationsstation,		enTypeOfBacNetTextListIn := enTypeOfBacNetTextList.ENDING		),	'M_NC_193')));
	M_NC_193._sDescription	:= 	fcUtfToAscii(Standard.CONCAT(	OBJ_NAME_DESCRIPTION,	fcGetBcText(	GVL_BACNET.fbBacNetParameter.metGetTextListName(enTypeOfBacNetFunktionIn := enTypeOfBacNetFunktion.Type_Automationsstation,		enTypeOfBacNetTextListIn := enTypeOfBacNetTextList.DESCRIPTION	),	'M_NC_193')));
	(* Create Id from Base Id and Object Nr (Last nummber of Name *)	
	M_NC_193.Create(diInstance := 193);
	(* Check if Created *)
	IF M_NC_193.xIsCreated THEN
		(* Set Group *)
		M_NC_193.setPropertyGroup(WagoTypesBacNet.eBACnetPropertyIdentifier.PROP_DESCRIPTION							,WagoTypesBacNet.eBACnetPropertyUpdateGroup.GROUP_CYCLIC);
		
		(* Set Ack Req *)
		M_NC_193.IAckRequired.xToOffNormal	:= FALSE;
		M_NC_193.IAckRequired.xToFault		:= TRUE;
		M_NC_193.IAckRequired.xToNormal		:= FALSE;
		
		(* Ziel												UTF8->ASCII		BacNet Text		Textlistname									BacNet Funktion																	BacNet Textlist type												TextId		*)
		M_NC_193.IEventMessageTextsConfig.sToOffNormal	:=	fcUtfToAscii(	fcGetBcText(	GVL_BACNET.fbBacNetParameter.metGetTextListName(enTypeOfBacNetFunktionIn := enTypeOfBacNetFunktion.Type_Automationsstation,		enTypeOfBacNetTextListIn := enTypeOfBacNetTextList.EVENTMESSAGE	),	'M_NC_193_ToOffNormal'	));		
		M_NC_193.IEventMessageTextsConfig.sToFault		:=	fcUtfToAscii(	fcGetBcText(	GVL_BACNET.fbBacNetParameter.metGetTextListName(enTypeOfBacNetFunktionIn := enTypeOfBacNetFunktion.Type_Automationsstation,		enTypeOfBacNetTextListIn := enTypeOfBacNetTextList.EVENTMESSAGE	),	'M_NC_193_ToFault'		));		
		M_NC_193.IEventMessageTextsConfig.sToNormal		:=	fcUtfToAscii(	fcGetBcText(	GVL_BACNET.fbBacNetParameter.metGetTextListName(enTypeOfBacNetFunktionIn := enTypeOfBacNetFunktion.Type_Automationsstation,		enTypeOfBacNetTextListIn := enTypeOfBacNetTextList.EVENTMESSAGE	),	'M_NC_193_ToNormal'		));		
		
		(* Notification Class & Type *)
		M_NC_193.udiNotificationClass					:=  193;	
		M_NC_193.eNotifyType							:= 	WagoTypesBACnet.eBACnetNotifyType.NOTIFY_TYPE_EVENT;
		(* Ziel												Convert			BacNet Text		Textlistname									BacNet Funktion																	BacNet Textlist type												TextId		*)	
		M_NC_193.IPriority.usiToOffNormal				:= 	TO_USINT(fcUtfToAscii(	fcGetBcText(	GVL_BACNET.fbBacNetParameter.metGetTextListName(enTypeOfBacNetFunktionIn := enTypeOfBacNetFunktion.Type_Automationsstation,		enTypeOfBacNetTextListIn := enTypeOfBacNetTextList.NC	),	'M_NC_193_Prio_ToOffNormal'	)));	
		M_NC_193.IPriority.usiToFault					:= 	TO_USINT(fcUtfToAscii(	fcGetBcText(	GVL_BACNET.fbBacNetParameter.metGetTextListName(enTypeOfBacNetFunktionIn := enTypeOfBacNetFunktion.Type_Automationsstation,		enTypeOfBacNetTextListIn := enTypeOfBacNetTextList.NC	),	'M_NC_193_Prio_ToFault'		)));	
		M_NC_193.IPriority.usiToNormal					:= 	TO_USINT(fcUtfToAscii(	fcGetBcText(	GVL_BACNET.fbBacNetParameter.metGetTextListName(enTypeOfBacNetFunktionIn := enTypeOfBacNetFunktion.Type_Automationsstation,		enTypeOfBacNetTextListIn := enTypeOfBacNetTextList.NC	),	'M_NC_193_Prio_ToNormal'		)));	
		
	ELSE
		M_NC_193.Delete();
	END_IF;
	(* Get Status *)
	metCreate_M_NC_193 := M_NC_193.xIsCreated;	
END_IF;
END_METHOD

METHOD metCreate_N_NC_224 : BOOL

VAR

END_VAR
(* N_NC_224*)
IF NOT N_NC_224.xIsCreated THEN
	(* Ziel						UTF8->ASCII						OBJ_NAME_BASE			BacNet Text		Textlistname									BacNet Funktion																	BacNet Textlist type												TextId		*)
	N_NC_224._sObjectName		:=	fcUtfToAscii(Standard.CONCAT(	OBJ_NAME_BASE		,	fcGetBcText(	GVL_BACNET.fbBacNetParameter.metGetTextListName(enTypeOfBacNetFunktionIn := enTypeOfBacNetFunktion.Type_Automationsstation,		enTypeOfBacNetTextListIn := enTypeOfBacNetTextList.ENDING		),	'N_NC_224')));
	N_NC_224._sDescription	:= 	fcUtfToAscii(Standard.CONCAT(	OBJ_NAME_DESCRIPTION,	fcGetBcText(	GVL_BACNET.fbBacNetParameter.metGetTextListName(enTypeOfBacNetFunktionIn := enTypeOfBacNetFunktion.Type_Automationsstation,		enTypeOfBacNetTextListIn := enTypeOfBacNetTextList.DESCRIPTION	),	'N_NC_224')));
	(* Create Id from Base Id and Object Nr (Last nummber of Name *)	
	N_NC_224.Create(diInstance := 224);
	(* Check if Created *)
	IF N_NC_224.xIsCreated THEN
		(* Set Group *)
		N_NC_224.setPropertyGroup(WagoTypesBacNet.eBACnetPropertyIdentifier.PROP_DESCRIPTION							,WagoTypesBacNet.eBACnetPropertyUpdateGroup.GROUP_CYCLIC);
		
		(* Set Ack Req *)
		N_NC_224.IAckRequired.xToOffNormal	:= FALSE;
		N_NC_224.IAckRequired.xToFault		:= FALSE;
		N_NC_224.IAckRequired.xToNormal		:= FALSE;
		
		(* Ziel												UTF8->ASCII		BacNet Text		Textlistname									BacNet Funktion																	BacNet Textlist type												TextId		*)
		N_NC_224.IEventMessageTextsConfig.sToOffNormal	:=	fcUtfToAscii(	fcGetBcText(	GVL_BACNET.fbBacNetParameter.metGetTextListName(enTypeOfBacNetFunktionIn := enTypeOfBacNetFunktion.Type_Automationsstation,		enTypeOfBacNetTextListIn := enTypeOfBacNetTextList.EVENTMESSAGE	),	'N_NC_224_ToOffNormal'	));		
		N_NC_224.IEventMessageTextsConfig.sToFault		:=	fcUtfToAscii(	fcGetBcText(	GVL_BACNET.fbBacNetParameter.metGetTextListName(enTypeOfBacNetFunktionIn := enTypeOfBacNetFunktion.Type_Automationsstation,		enTypeOfBacNetTextListIn := enTypeOfBacNetTextList.EVENTMESSAGE	),	'N_NC_224_ToFault'		));		
		N_NC_224.IEventMessageTextsConfig.sToNormal		:=	fcUtfToAscii(	fcGetBcText(	GVL_BACNET.fbBacNetParameter.metGetTextListName(enTypeOfBacNetFunktionIn := enTypeOfBacNetFunktion.Type_Automationsstation,		enTypeOfBacNetTextListIn := enTypeOfBacNetTextList.EVENTMESSAGE	),	'N_NC_224_ToNormal'		));		
		
		(* Notification Class & Type *)
		N_NC_224.udiNotificationClass					:=  224;	
		N_NC_224.eNotifyType							:= 	WagoTypesBACnet.eBACnetNotifyType.NOTIFY_TYPE_EVENT;
		(* Ziel												Convert			BacNet Text		Textlistname									BacNet Funktion																	BacNet Textlist type												TextId		*)	
		N_NC_224.IPriority.usiToOffNormal				:= 	TO_USINT(fcUtfToAscii(	fcGetBcText(	GVL_BACNET.fbBacNetParameter.metGetTextListName(enTypeOfBacNetFunktionIn := enTypeOfBacNetFunktion.Type_Automationsstation,		enTypeOfBacNetTextListIn := enTypeOfBacNetTextList.NC	),	'N_NC_224_Prio_ToOffNormal'	)));	
		N_NC_224.IPriority.usiToFault					:= 	TO_USINT(fcUtfToAscii(	fcGetBcText(	GVL_BACNET.fbBacNetParameter.metGetTextListName(enTypeOfBacNetFunktionIn := enTypeOfBacNetFunktion.Type_Automationsstation,		enTypeOfBacNetTextListIn := enTypeOfBacNetTextList.NC	),	'N_NC_224_Prio_ToFault'		)));	
		N_NC_224.IPriority.usiToNormal					:= 	TO_USINT(fcUtfToAscii(	fcGetBcText(	GVL_BACNET.fbBacNetParameter.metGetTextListName(enTypeOfBacNetFunktionIn := enTypeOfBacNetFunktion.Type_Automationsstation,		enTypeOfBacNetTextListIn := enTypeOfBacNetTextList.NC	),	'N_NC_224_Prio_ToNormal'		)));	
		
	ELSE
		N_NC_224.Delete();
	END_IF;
	(* Get Status *)
	metCreate_N_NC_224 := N_NC_224.xIsCreated;	
END_IF;
END_METHOD

METHOD metCreate_N_NC_225 : BOOL

VAR

END_VAR
(* N_NC_225*)
IF NOT N_NC_225.xIsCreated THEN
	(* Ziel						UTF8->ASCII						OBJ_NAME_BASE			BacNet Text		Textlistname									BacNet Funktion																	BacNet Textlist type												TextId		*)
	N_NC_225._sObjectName		:=	fcUtfToAscii(Standard.CONCAT(	OBJ_NAME_BASE		,	fcGetBcText(	GVL_BACNET.fbBacNetParameter.metGetTextListName(enTypeOfBacNetFunktionIn := enTypeOfBacNetFunktion.Type_Automationsstation,		enTypeOfBacNetTextListIn := enTypeOfBacNetTextList.ENDING		),	'N_NC_225')));
	N_NC_225._sDescription	:= 	fcUtfToAscii(Standard.CONCAT(	OBJ_NAME_DESCRIPTION,	fcGetBcText(	GVL_BACNET.fbBacNetParameter.metGetTextListName(enTypeOfBacNetFunktionIn := enTypeOfBacNetFunktion.Type_Automationsstation,		enTypeOfBacNetTextListIn := enTypeOfBacNetTextList.DESCRIPTION	),	'N_NC_225')));
	(* Create Id from Base Id and Object Nr (Last nummber of Name *)	
	N_NC_225.Create(diInstance := 225);
	(* Check if Created *)
	IF N_NC_225.xIsCreated THEN
		(* Set Group *)
		N_NC_225.setPropertyGroup(WagoTypesBacNet.eBACnetPropertyIdentifier.PROP_DESCRIPTION							,WagoTypesBacNet.eBACnetPropertyUpdateGroup.GROUP_CYCLIC);
		
		(* Set Ack Req *)
		N_NC_225.IAckRequired.xToOffNormal	:= FALSE;
		N_NC_225.IAckRequired.xToFault		:= TRUE;
		N_NC_225.IAckRequired.xToNormal		:= FALSE;
		
		(* Ziel												UTF8->ASCII		BacNet Text		Textlistname									BacNet Funktion																	BacNet Textlist type												TextId		*)
		N_NC_225.IEventMessageTextsConfig.sToOffNormal	:=	fcUtfToAscii(	fcGetBcText(	GVL_BACNET.fbBacNetParameter.metGetTextListName(enTypeOfBacNetFunktionIn := enTypeOfBacNetFunktion.Type_Automationsstation,		enTypeOfBacNetTextListIn := enTypeOfBacNetTextList.EVENTMESSAGE	),	'N_NC_225_ToOffNormal'	));		
		N_NC_225.IEventMessageTextsConfig.sToFault		:=	fcUtfToAscii(	fcGetBcText(	GVL_BACNET.fbBacNetParameter.metGetTextListName(enTypeOfBacNetFunktionIn := enTypeOfBacNetFunktion.Type_Automationsstation,		enTypeOfBacNetTextListIn := enTypeOfBacNetTextList.EVENTMESSAGE	),	'N_NC_225_ToFault'		));		
		N_NC_225.IEventMessageTextsConfig.sToNormal		:=	fcUtfToAscii(	fcGetBcText(	GVL_BACNET.fbBacNetParameter.metGetTextListName(enTypeOfBacNetFunktionIn := enTypeOfBacNetFunktion.Type_Automationsstation,		enTypeOfBacNetTextListIn := enTypeOfBacNetTextList.EVENTMESSAGE	),	'N_NC_225_ToNormal'		));		
		
		(* Notification Class & Type *)
		N_NC_225.udiNotificationClass					:=  225;	
		N_NC_225.eNotifyType							:= 	WagoTypesBACnet.eBACnetNotifyType.NOTIFY_TYPE_EVENT;
		(* Ziel												Convert			BacNet Text		Textlistname									BacNet Funktion																	BacNet Textlist type												TextId		*)	
		N_NC_225.IPriority.usiToOffNormal				:= 	TO_USINT(fcUtfToAscii(	fcGetBcText(	GVL_BACNET.fbBacNetParameter.metGetTextListName(enTypeOfBacNetFunktionIn := enTypeOfBacNetFunktion.Type_Automationsstation,		enTypeOfBacNetTextListIn := enTypeOfBacNetTextList.NC	),	'N_NC_225_Prio_ToOffNormal'	)));	
		N_NC_225.IPriority.usiToFault					:= 	TO_USINT(fcUtfToAscii(	fcGetBcText(	GVL_BACNET.fbBacNetParameter.metGetTextListName(enTypeOfBacNetFunktionIn := enTypeOfBacNetFunktion.Type_Automationsstation,		enTypeOfBacNetTextListIn := enTypeOfBacNetTextList.NC	),	'N_NC_225_Prio_ToFault'		)));	
		N_NC_225.IPriority.usiToNormal					:= 	TO_USINT(fcUtfToAscii(	fcGetBcText(	GVL_BACNET.fbBacNetParameter.metGetTextListName(enTypeOfBacNetFunktionIn := enTypeOfBacNetFunktion.Type_Automationsstation,		enTypeOfBacNetTextListIn := enTypeOfBacNetTextList.NC	),	'N_NC_225_Prio_ToNormal'		)));	
		
	ELSE
		N_NC_225.Delete();
	END_IF;
	(* Get Status *)
	metCreate_N_NC_225 := N_NC_225.xIsCreated;	
END_IF;
END_METHOD

METHOD metCreate_O_BV_1 : BOOL
(* O_BV_1*)
IF NOT O_BV_1.xIsCreated THEN
	(* Ziel						UTF8->ASCII						OBJ_NAME_BASE			BacNet Text		Textlistname									BacNet Funktion																BacNet Textlist type												TextId		*)
	O_BV_1._sObjectName		:=	fcUtfToAscii(Standard.CONCAT(	OBJ_NAME_BASE		,	fcGetBcText(	GVL_BACNET.fbBacNetParameter.metGetTextListName(enTypeOfBacNetFunktionIn := enTypeOfBacNetFunktion.Type_Automationsstation,		enTypeOfBacNetTextListIn := enTypeOfBacNetTextList.ENDING		),	'O_BV_1')));
	O_BV_1._sDescription	:= 	fcUtfToAscii(Standard.CONCAT(	OBJ_NAME_DESCRIPTION,	fcGetBcText(	GVL_BACNET.fbBacNetParameter.metGetTextListName(enTypeOfBacNetFunktionIn := enTypeOfBacNetFunktion.Type_Automationsstation,		enTypeOfBacNetTextListIn := enTypeOfBacNetTextList.DESCRIPTION	),	'O_BV_1')));
	(* Create Id from Base Id and Object Nr (Last nummber of Name *)	
	O_BV_1.Create(diInstance := TO_DINT(Standard.CONCAT(TO_STRING(dwOBJ_ID_BASE),'1')));
	(* Check if Created *)
	IF O_BV_1.xIsCreated THEN
		(* Set Group *)
		O_BV_1.setPropertyGroup(WagoTypesBacNet.eBACnetPropertyIdentifier.PROP_PRESENT_VALUE						,WagoTypesBacNet.eBACnetPropertyUpdateGroup.GROUP_CYCLIC);
		O_BV_1.setPropertyGroup(WagoTypesBacNet.eBACnetPropertyIdentifier.PROP_PRIORITY_ARRAY						,WagoTypesBacNet.eBACnetPropertyUpdateGroup.GROUP_CYCLIC);
		O_BV_1.setPropertyGroup(WagoTypesBacNet.eBACnetPropertyIdentifier.PROP_ELAPSED_ACTIVE_TIME					,WagoTypesBacNet.eBACnetPropertyUpdateGroup.GROUP_CYCLIC);
		O_BV_1.setPropertyGroup(WagoTypesBacNet.eBACnetPropertyIdentifier.PROP_DESCRIPTION							,WagoTypesBacNet.eBACnetPropertyUpdateGroup.GROUP_CYCLIC);
		O_BV_1.setPropertyGroup(WagoTypesBacNet.eBACnetPropertyIdentifier.PROP_EVENT_MESSAGE_TEXTS_CONFIG			,WagoTypesBacNet.eBACnetPropertyUpdateGroup.GROUP_CYCLIC);
		(* Set Description to Overwrite retain*)
		O_BV_1.sDescription	:= O_BV_1._sDescription;
		(* Ziel												UTF8->ASCII		BacNet Text		Textlistname									BacNet Funktion																BacNet Textlist type												TextId		*)
		O_BV_1.IEventMessageTextsConfig.sToOffNormal	:=	fcUtfToAscii(	fcGetBcText(	GVL_BACNET.fbBacNetParameter.metGetTextListName(enTypeOfBacNetFunktionIn := enTypeOfBacNetFunktion.Type_Automationsstation,		enTypeOfBacNetTextListIn := enTypeOfBacNetTextList.EVENTMESSAGE	),	'O_BV_1_ToOffNormal'	));		
		O_BV_1.IEventMessageTextsConfig.sToFault		:=	fcUtfToAscii(	fcGetBcText(	GVL_BACNET.fbBacNetParameter.metGetTextListName(enTypeOfBacNetFunktionIn := enTypeOfBacNetFunktion.Type_Automationsstation,		enTypeOfBacNetTextListIn := enTypeOfBacNetTextList.EVENTMESSAGE	),	'O_BV_1_ToFault'		));		
		O_BV_1.IEventMessageTextsConfig.sToNormal		:=	fcUtfToAscii(	fcGetBcText(	GVL_BACNET.fbBacNetParameter.metGetTextListName(enTypeOfBacNetFunktionIn := enTypeOfBacNetFunktion.Type_Automationsstation,		enTypeOfBacNetTextListIn := enTypeOfBacNetTextList.EVENTMESSAGE	),	'O_BV_1_ToNormal'		));		

		(* Ziel												UTF8->ASCII		BacNet Text		Textlistname									BacNet Funktion																BacNet Textlist type												TextId		*)	
		O_BV_1.sActiveText								:= 	fcUtfToAscii(	fcGetBcText(	GVL_BACNET.fbBacNetParameter.metGetTextListName(enTypeOfBacNetFunktionIn := enTypeOfBacNetFunktion.Type_Automationsstation,		enTypeOfBacNetTextListIn := enTypeOfBacNetTextList.PRESENTVALUE	),	'O_BV_1_ST_ACTIVE'		));
		O_BV_1.sInactiveText							:= 	fcUtfToAscii(	fcGetBcText(	GVL_BACNET.fbBacNetParameter.metGetTextListName(enTypeOfBacNetFunktionIn := enTypeOfBacNetFunktion.Type_Automationsstation,		enTypeOfBacNetTextListIn := enTypeOfBacNetTextList.PRESENTVALUE	),	'O_BV_1_ST_INACTIVE'	));	

		(* Ziel												Convert			BacNet Text		Textlistname									BacNet Funktion																	BacNet Textlist type												TextId		*)	
		O_BV_1.udiNotificationClass						:= 	TO_UDINT	(	fcGetBcText(	GVL_BACNET.fbBacNetParameter.metGetTextListName(enTypeOfBacNetFunktionIn := enTypeOfBacNetFunktion.Type_Automationsstation,		enTypeOfBacNetTextListIn := enTypeOfBacNetTextList.NC			),	'O_BV_1_NC'	));	
		O_BV_1.eNotifyType								:= 	WagoTypesBACnet.eBACnetNotifyType.NOTIFY_TYPE_ALARM;		
		O_BV_1.xAlarmValue								:= 	TO_BOOL		(	fcGetBcText(	GVL_BACNET.fbBacNetParameter.metGetTextListName(enTypeOfBacNetFunktionIn := enTypeOfBacNetFunktion.Type_Automationsstation,		enTypeOfBacNetTextListIn := enTypeOfBacNetTextList.NC			),	'O_BV_1_ALV'	));	
		
	ELSE
		O_BV_1.Delete();
	END_IF;
	(* Get Status *)
	metCreate_O_BV_1 := O_BV_1.xIsCreated;	
END_IF;
END_METHOD

METHOD metCreate_P_BV_2 : BOOL
(* P_BV_2*)
IF NOT P_BV_2.xIsCreated THEN
	(* Ziel						UTF8->ASCII						OBJ_NAME_BASE			BacNet Text		Textlistname									BacNet Funktion																BacNet Textlist type												TextId		*)
	P_BV_2._sObjectName		:=	fcUtfToAscii(Standard.CONCAT(	OBJ_NAME_BASE		,	fcGetBcText(	GVL_BACNET.fbBacNetParameter.metGetTextListName(enTypeOfBacNetFunktionIn := enTypeOfBacNetFunktion.Type_Automationsstation,		enTypeOfBacNetTextListIn := enTypeOfBacNetTextList.ENDING		),	'P_BV_2')));
	P_BV_2._sDescription	:= 	fcUtfToAscii(Standard.CONCAT(	OBJ_NAME_DESCRIPTION,	fcGetBcText(	GVL_BACNET.fbBacNetParameter.metGetTextListName(enTypeOfBacNetFunktionIn := enTypeOfBacNetFunktion.Type_Automationsstation,		enTypeOfBacNetTextListIn := enTypeOfBacNetTextList.DESCRIPTION	),	'P_BV_2')));
	(* Create Id from Base Id and Object Nr (Last nummber of Name *)	
	P_BV_2.Create(diInstance := TO_DINT(Standard.CONCAT(TO_STRING(dwOBJ_ID_BASE),'2')));
	(* Check if Created *)
	IF P_BV_2.xIsCreated THEN
		(* Set Group *)
		P_BV_2.setPropertyGroup(WagoTypesBacNet.eBACnetPropertyIdentifier.PROP_PRESENT_VALUE						,WagoTypesBacNet.eBACnetPropertyUpdateGroup.GROUP_CYCLIC);
		P_BV_2.setPropertyGroup(WagoTypesBacNet.eBACnetPropertyIdentifier.PROP_PRIORITY_ARRAY						,WagoTypesBacNet.eBACnetPropertyUpdateGroup.GROUP_CYCLIC);
		P_BV_2.setPropertyGroup(WagoTypesBacNet.eBACnetPropertyIdentifier.PROP_ELAPSED_ACTIVE_TIME					,WagoTypesBacNet.eBACnetPropertyUpdateGroup.GROUP_CYCLIC);
		P_BV_2.setPropertyGroup(WagoTypesBacNet.eBACnetPropertyIdentifier.PROP_DESCRIPTION							,WagoTypesBacNet.eBACnetPropertyUpdateGroup.GROUP_CYCLIC);
		P_BV_2.setPropertyGroup(WagoTypesBacNet.eBACnetPropertyIdentifier.PROP_EVENT_MESSAGE_TEXTS_CONFIG			,WagoTypesBacNet.eBACnetPropertyUpdateGroup.GROUP_CYCLIC);
		(* Set Description to Overwrite retain*)
		P_BV_2.sDescription	:= P_BV_2._sDescription;
		(* Ziel												UTF8->ASCII		BacNet Text		Textlistname									BacNet Funktion																BacNet Textlist type												TextId		*)
		P_BV_2.IEventMessageTextsConfig.sToOffNormal	:=	fcUtfToAscii(	fcGetBcText(	GVL_BACNET.fbBacNetParameter.metGetTextListName(enTypeOfBacNetFunktionIn := enTypeOfBacNetFunktion.Type_Automationsstation,		enTypeOfBacNetTextListIn := enTypeOfBacNetTextList.EVENTMESSAGE	),	'P_BV_2_ToOffNormal'	));		
		P_BV_2.IEventMessageTextsConfig.sToFault		:=	fcUtfToAscii(	fcGetBcText(	GVL_BACNET.fbBacNetParameter.metGetTextListName(enTypeOfBacNetFunktionIn := enTypeOfBacNetFunktion.Type_Automationsstation,		enTypeOfBacNetTextListIn := enTypeOfBacNetTextList.EVENTMESSAGE	),	'P_BV_2_ToFault'		));		
		P_BV_2.IEventMessageTextsConfig.sToNormal		:=	fcUtfToAscii(	fcGetBcText(	GVL_BACNET.fbBacNetParameter.metGetTextListName(enTypeOfBacNetFunktionIn := enTypeOfBacNetFunktion.Type_Automationsstation,		enTypeOfBacNetTextListIn := enTypeOfBacNetTextList.EVENTMESSAGE	),	'P_BV_2_ToNormal'		));		

		(* Ziel												UTF8->ASCII		BacNet Text		Textlistname									BacNet Funktion																BacNet Textlist type												TextId		*)	
		P_BV_2.sActiveText								:= 	fcUtfToAscii(	fcGetBcText(	GVL_BACNET.fbBacNetParameter.metGetTextListName(enTypeOfBacNetFunktionIn := enTypeOfBacNetFunktion.Type_Automationsstation,		enTypeOfBacNetTextListIn := enTypeOfBacNetTextList.PRESENTVALUE	),	'P_BV_2_ST_ACTIVE'		));
		P_BV_2.sInactiveText							:= 	fcUtfToAscii(	fcGetBcText(	GVL_BACNET.fbBacNetParameter.metGetTextListName(enTypeOfBacNetFunktionIn := enTypeOfBacNetFunktion.Type_Automationsstation,		enTypeOfBacNetTextListIn := enTypeOfBacNetTextList.PRESENTVALUE	),	'P_BV_2_ST_INACTIVE'	));	

		(* Ziel												Convert			BacNet Text		Textlistname									BacNet Funktion																	BacNet Textlist type												TextId		*)	
		P_BV_2.udiNotificationClass						:= 	TO_UDINT	(	fcGetBcText(	GVL_BACNET.fbBacNetParameter.metGetTextListName(enTypeOfBacNetFunktionIn := enTypeOfBacNetFunktion.Type_Automationsstation,		enTypeOfBacNetTextListIn := enTypeOfBacNetTextList.NC			),	'P_BV_2_NC'	));	
		P_BV_2.eNotifyType								:= 	WagoTypesBACnet.eBACnetNotifyType.NOTIFY_TYPE_ALARM;		
		P_BV_2.xAlarmValue								:= 	TO_BOOL		(	fcGetBcText(	GVL_BACNET.fbBacNetParameter.metGetTextListName(enTypeOfBacNetFunktionIn := enTypeOfBacNetFunktion.Type_Automationsstation,		enTypeOfBacNetTextListIn := enTypeOfBacNetTextList.NC			),	'P_BV_2_ALV'	));	
		
	ELSE
		P_BV_2.Delete();
	END_IF;
	(* Get Status *)
	metCreate_P_BV_2 := P_BV_2.xIsCreated;	
END_IF;
END_METHOD

METHOD metCreate_Q_BV_3 : BOOL
(* Q_BV_3*)
IF NOT Q_BV_3.xIsCreated THEN
	(* Ziel						UTF8->ASCII						OBJ_NAME_BASE			BacNet Text		Textlistname									BacNet Funktion																BacNet Textlist type												TextId		*)
	Q_BV_3._sObjectName		:=	fcUtfToAscii(Standard.CONCAT(	OBJ_NAME_BASE		,	fcGetBcText(	GVL_BACNET.fbBacNetParameter.metGetTextListName(enTypeOfBacNetFunktionIn := enTypeOfBacNetFunktion.Type_Automationsstation,		enTypeOfBacNetTextListIn := enTypeOfBacNetTextList.ENDING		),	'Q_BV_3')));
	Q_BV_3._sDescription	:= 	fcUtfToAscii(Standard.CONCAT(	OBJ_NAME_DESCRIPTION,	fcGetBcText(	GVL_BACNET.fbBacNetParameter.metGetTextListName(enTypeOfBacNetFunktionIn := enTypeOfBacNetFunktion.Type_Automationsstation,		enTypeOfBacNetTextListIn := enTypeOfBacNetTextList.DESCRIPTION	),	'Q_BV_3')));
	(* Create Id from Base Id and Object Nr (Last nummber of Name *)	
	Q_BV_3.Create(diInstance := TO_DINT(Standard.CONCAT(TO_STRING(dwOBJ_ID_BASE),'3')));
	(* Check if Created *)
	IF Q_BV_3.xIsCreated THEN
		(* Set Group *)
		Q_BV_3.setPropertyGroup(WagoTypesBacNet.eBACnetPropertyIdentifier.PROP_PRESENT_VALUE						,WagoTypesBacNet.eBACnetPropertyUpdateGroup.GROUP_CYCLIC);
		Q_BV_3.setPropertyGroup(WagoTypesBacNet.eBACnetPropertyIdentifier.PROP_PRIORITY_ARRAY						,WagoTypesBacNet.eBACnetPropertyUpdateGroup.GROUP_CYCLIC);
		Q_BV_3.setPropertyGroup(WagoTypesBacNet.eBACnetPropertyIdentifier.PROP_ELAPSED_ACTIVE_TIME					,WagoTypesBacNet.eBACnetPropertyUpdateGroup.GROUP_CYCLIC);
		Q_BV_3.setPropertyGroup(WagoTypesBacNet.eBACnetPropertyIdentifier.PROP_DESCRIPTION							,WagoTypesBacNet.eBACnetPropertyUpdateGroup.GROUP_CYCLIC);
		Q_BV_3.setPropertyGroup(WagoTypesBacNet.eBACnetPropertyIdentifier.PROP_EVENT_MESSAGE_TEXTS_CONFIG			,WagoTypesBacNet.eBACnetPropertyUpdateGroup.GROUP_CYCLIC);
		(* Set Description to Overwrite retain*)
		Q_BV_3.sDescription	:= Q_BV_3._sDescription;
		(* Ziel												UTF8->ASCII		BacNet Text		Textlistname									BacNet Funktion																BacNet Textlist type												TextId		*)
		Q_BV_3.IEventMessageTextsConfig.sToOffNormal	:=	fcUtfToAscii(	fcGetBcText(	GVL_BACNET.fbBacNetParameter.metGetTextListName(enTypeOfBacNetFunktionIn := enTypeOfBacNetFunktion.Type_Automationsstation,		enTypeOfBacNetTextListIn := enTypeOfBacNetTextList.EVENTMESSAGE	),	'Q_BV_3_ToOffNormal'	));		
		Q_BV_3.IEventMessageTextsConfig.sToFault		:=	fcUtfToAscii(	fcGetBcText(	GVL_BACNET.fbBacNetParameter.metGetTextListName(enTypeOfBacNetFunktionIn := enTypeOfBacNetFunktion.Type_Automationsstation,		enTypeOfBacNetTextListIn := enTypeOfBacNetTextList.EVENTMESSAGE	),	'Q_BV_3_ToFault'		));		
		Q_BV_3.IEventMessageTextsConfig.sToNormal		:=	fcUtfToAscii(	fcGetBcText(	GVL_BACNET.fbBacNetParameter.metGetTextListName(enTypeOfBacNetFunktionIn := enTypeOfBacNetFunktion.Type_Automationsstation,		enTypeOfBacNetTextListIn := enTypeOfBacNetTextList.EVENTMESSAGE	),	'Q_BV_3_ToNormal'		));		

		(* Ziel												UTF8->ASCII		BacNet Text		Textlistname									BacNet Funktion																BacNet Textlist type												TextId		*)	
		Q_BV_3.sActiveText								:= 	fcUtfToAscii(	fcGetBcText(	GVL_BACNET.fbBacNetParameter.metGetTextListName(enTypeOfBacNetFunktionIn := enTypeOfBacNetFunktion.Type_Automationsstation,		enTypeOfBacNetTextListIn := enTypeOfBacNetTextList.PRESENTVALUE	),	'Q_BV_3_ST_ACTIVE'		));
		Q_BV_3.sInactiveText							:= 	fcUtfToAscii(	fcGetBcText(	GVL_BACNET.fbBacNetParameter.metGetTextListName(enTypeOfBacNetFunktionIn := enTypeOfBacNetFunktion.Type_Automationsstation,		enTypeOfBacNetTextListIn := enTypeOfBacNetTextList.PRESENTVALUE	),	'Q_BV_3_ST_INACTIVE'	));	

		(* Ziel												Convert			BacNet Text		Textlistname									BacNet Funktion																	BacNet Textlist type												TextId		*)	
		Q_BV_3.udiNotificationClass						:= 	TO_UDINT	(	fcGetBcText(	GVL_BACNET.fbBacNetParameter.metGetTextListName(enTypeOfBacNetFunktionIn := enTypeOfBacNetFunktion.Type_Automationsstation,		enTypeOfBacNetTextListIn := enTypeOfBacNetTextList.NC			),	'Q_BV_3_NC'	));	
		Q_BV_3.eNotifyType								:= 	WagoTypesBACnet.eBACnetNotifyType.NOTIFY_TYPE_ALARM;		
		Q_BV_3.xAlarmValue								:= 	TO_BOOL		(	fcGetBcText(	GVL_BACNET.fbBacNetParameter.metGetTextListName(enTypeOfBacNetFunktionIn := enTypeOfBacNetFunktion.Type_Automationsstation,		enTypeOfBacNetTextListIn := enTypeOfBacNetTextList.NC			),	'Q_BV_3_ALV'	));	
		
	ELSE
		Q_BV_3.Delete();
	END_IF;
	(* Get Status *)
	metCreate_Q_BV_3 := Q_BV_3.xIsCreated;	
END_IF;
END_METHOD

METHOD metCreate_R_BV_4 : BOOL
(* R_BV_4*)
IF NOT R_BV_4.xIsCreated THEN
	(* Ziel						UTF8->ASCII						OBJ_NAME_BASE			BacNet Text		Textlistname									BacNet Funktion																BacNet Textlist type												TextId		*)
	R_BV_4._sObjectName		:=	fcUtfToAscii(Standard.CONCAT(	OBJ_NAME_BASE		,	fcGetBcText(	GVL_BACNET.fbBacNetParameter.metGetTextListName(enTypeOfBacNetFunktionIn := enTypeOfBacNetFunktion.Type_Automationsstation,		enTypeOfBacNetTextListIn := enTypeOfBacNetTextList.ENDING		),	'R_BV_4')));
	R_BV_4._sDescription	:= 	fcUtfToAscii(Standard.CONCAT(	OBJ_NAME_DESCRIPTION,	fcGetBcText(	GVL_BACNET.fbBacNetParameter.metGetTextListName(enTypeOfBacNetFunktionIn := enTypeOfBacNetFunktion.Type_Automationsstation,		enTypeOfBacNetTextListIn := enTypeOfBacNetTextList.DESCRIPTION	),	'R_BV_4')));
	(* Create Id from Base Id and Object Nr (Last nummber of Name *)	
	R_BV_4.Create(diInstance := TO_DINT(Standard.CONCAT(TO_STRING(dwOBJ_ID_BASE),'4')));
	(* Check if Created *)
	IF R_BV_4.xIsCreated THEN
		(* Set Group *)
		R_BV_4.setPropertyGroup(WagoTypesBacNet.eBACnetPropertyIdentifier.PROP_PRESENT_VALUE						,WagoTypesBacNet.eBACnetPropertyUpdateGroup.GROUP_CYCLIC);
		R_BV_4.setPropertyGroup(WagoTypesBacNet.eBACnetPropertyIdentifier.PROP_PRIORITY_ARRAY						,WagoTypesBacNet.eBACnetPropertyUpdateGroup.GROUP_CYCLIC);
		R_BV_4.setPropertyGroup(WagoTypesBacNet.eBACnetPropertyIdentifier.PROP_ELAPSED_ACTIVE_TIME					,WagoTypesBacNet.eBACnetPropertyUpdateGroup.GROUP_CYCLIC);
		R_BV_4.setPropertyGroup(WagoTypesBacNet.eBACnetPropertyIdentifier.PROP_DESCRIPTION							,WagoTypesBacNet.eBACnetPropertyUpdateGroup.GROUP_CYCLIC);
		R_BV_4.setPropertyGroup(WagoTypesBacNet.eBACnetPropertyIdentifier.PROP_EVENT_MESSAGE_TEXTS_CONFIG			,WagoTypesBacNet.eBACnetPropertyUpdateGroup.GROUP_CYCLIC);
		(* Set Description to Overwrite retain*)
		R_BV_4.sDescription	:= R_BV_4._sDescription;
		(* Ziel												UTF8->ASCII		BacNet Text		Textlistname									BacNet Funktion																BacNet Textlist type												TextId		*)
		R_BV_4.IEventMessageTextsConfig.sToOffNormal	:=	fcUtfToAscii(	fcGetBcText(	GVL_BACNET.fbBacNetParameter.metGetTextListName(enTypeOfBacNetFunktionIn := enTypeOfBacNetFunktion.Type_Automationsstation,		enTypeOfBacNetTextListIn := enTypeOfBacNetTextList.EVENTMESSAGE	),	'R_BV_4_ToOffNormal'	));		
		R_BV_4.IEventMessageTextsConfig.sToFault		:=	fcUtfToAscii(	fcGetBcText(	GVL_BACNET.fbBacNetParameter.metGetTextListName(enTypeOfBacNetFunktionIn := enTypeOfBacNetFunktion.Type_Automationsstation,		enTypeOfBacNetTextListIn := enTypeOfBacNetTextList.EVENTMESSAGE	),	'R_BV_4_ToFault'		));		
		R_BV_4.IEventMessageTextsConfig.sToNormal		:=	fcUtfToAscii(	fcGetBcText(	GVL_BACNET.fbBacNetParameter.metGetTextListName(enTypeOfBacNetFunktionIn := enTypeOfBacNetFunktion.Type_Automationsstation,		enTypeOfBacNetTextListIn := enTypeOfBacNetTextList.EVENTMESSAGE	),	'R_BV_4_ToNormal'		));		

		(* Ziel												UTF8->ASCII		BacNet Text		Textlistname									BacNet Funktion																BacNet Textlist type												TextId		*)	
		R_BV_4.sActiveText								:= 	fcUtfToAscii(	fcGetBcText(	GVL_BACNET.fbBacNetParameter.metGetTextListName(enTypeOfBacNetFunktionIn := enTypeOfBacNetFunktion.Type_Automationsstation,		enTypeOfBacNetTextListIn := enTypeOfBacNetTextList.PRESENTVALUE	),	'R_BV_4_ST_ACTIVE'		));
		R_BV_4.sInactiveText							:= 	fcUtfToAscii(	fcGetBcText(	GVL_BACNET.fbBacNetParameter.metGetTextListName(enTypeOfBacNetFunktionIn := enTypeOfBacNetFunktion.Type_Automationsstation,		enTypeOfBacNetTextListIn := enTypeOfBacNetTextList.PRESENTVALUE	),	'R_BV_4_ST_INACTIVE'	));	

		(* Ziel												Convert			BacNet Text		Textlistname									BacNet Funktion																	BacNet Textlist type												TextId		*)	
		R_BV_4.udiNotificationClass						:= 	TO_UDINT	(	fcGetBcText(	GVL_BACNET.fbBacNetParameter.metGetTextListName(enTypeOfBacNetFunktionIn := enTypeOfBacNetFunktion.Type_Automationsstation,		enTypeOfBacNetTextListIn := enTypeOfBacNetTextList.NC			),	'R_BV_4_NC'	));	
		R_BV_4.eNotifyType								:= 	WagoTypesBACnet.eBACnetNotifyType.NOTIFY_TYPE_EVENT;		
		R_BV_4.xAlarmValue								:= 	TO_BOOL		(	fcGetBcText(	GVL_BACNET.fbBacNetParameter.metGetTextListName(enTypeOfBacNetFunktionIn := enTypeOfBacNetFunktion.Type_Automationsstation,		enTypeOfBacNetTextListIn := enTypeOfBacNetTextList.NC			),	'R_BV_4_ALV'	));	
		
	ELSE
		R_BV_4.Delete();
	END_IF;
	(* Get Status *)
	metCreate_R_BV_4 := R_BV_4.xIsCreated;	
END_IF;
END_METHOD

